LIN {X 0,Y 143.834,Z 840.119,A -85,B 0,C 180,E1 -24449.132,E2 -24449.132} C_VEL
LIN {X 0,Y 144.282,Z 844.837,A -85,B 0,C 180,E1 -24453.998,E2 -24453.998} C_VEL
LIN {X 0,Y 145.051,Z 847.23,A -85,B 0,C 180,E1 -24457.193,E2 -24457.193} C_VEL
LIN {X 0,Y 147.333,Z 850.158,A -85,B 0,C 180,E1 -24462.562,E2 -24462.562} C_VEL
LIN {X 0,Y 150.85,Z 851.632,A -85,B 0,C 180,E1 -24468.065,E2 -24468.065} C_VEL
LIN {X 0,Y 155.654,Z 851.525,A -85,B 0,C 180,E1 -24473.384,E2 -24473.384} C_VEL
LIN {X 0,Y 161.705,Z 849.693,A -85,B 0,C 180,E1 -24478.445,E2 -24478.445} C_VEL
LIN {X 0,Y 168.926,Z 846.027,A -85,B 0,C 180,E1 -24483.134,E2 -24483.134} C_VEL
LIN {X 0,Y 175.939,Z 841.345,A -85,B 0,C 180,E1 -24486.882,E2 -24486.882} C_VEL
LIN {X 0,Y 182.747,Z 835.741,A -85,B 0,C 180,E1 -24489.966,E2 -24489.966} C_VEL
LIN {X 0,Y 184.593,Z 833.905,A -85,B 0,C 180,E1 -24490.974,E2 -24490.974} C_VEL
LIN {X 0,Y 185.748,Z 831.879,A -85,B 0,C 180,E1 -24493.121,E2 -24493.121} C_VEL
LIN {X 0,Y 186.699,Z 829.958,A -85,B 0,C 180,E1 -24495.278,E2 -24495.278} C_VEL
LIN {X 0,Y 186.772,Z 828.948,A -85,B 0,C 180,E1 -24497.519,E2 -24497.519} C_VEL
LIN {X 0,Y 186.523,Z 828.401,A -85,B 0,C 180,E1 -24499.823,E2 -24499.823} C_VEL
LIN {X 0,Y 186.294,Z 828.27,A -85,B 0,C 180,E1 -24502.164,E2 -24502.164} C_VEL
LIN {X 0,Y 185.911,Z 829.094,A -85,B 0,C 180,E1 -24506.977,E2 -24506.977} C_VEL
LIN {X 0,Y 185.613,Z 830.4,A -85,B 0,C 180,E1 -24509.487,E2 -24509.487} C_VEL
LIN {X 0,Y 185.359,Z 832.163,A -85,B 0,C 180,E1 -24512.061,E2 -24512.061} C_VEL
LIN {X 0,Y 184.447,Z 837.377,A -85,B 0,C 180,E1 -24516.853,E2 -24516.853} C_VEL
LIN {X 0,Y 183.603,Z 840.183,A -85,B 0,C 180,E1 -24518.656,E2 -24518.656} C_VEL
LIN {X 0,Y 178.489,Z 848.812,A -85,B 0,C 180,E1 -24522.398,E2 -24522.398} C_VEL
LIN {X 0,Y 172.641,Z 857.248,A -85,B 0,C 180,E1 -24526.207,E2 -24526.207} C_VEL
LIN {X 0,Y 167.309,Z 863.837,A -85,B 0,C 180,E1 -24529.478,E2 -24529.478} C_VEL
LIN {X 0,Y 160.39,Z 870.953,A -85,B 0,C 180,E1 -24533.733,E2 -24533.733} C_VEL
LIN {X 0,Y 155.765,Z 875.456,A -85,B 0,C 180,E1 -24537.218,E2 -24537.218} C_VEL
LIN {X 0,Y 150.033,Z 880.097,A -85,B 0,C 180,E1 -24542.067,E2 -24542.067} C_VEL
LIN {X 0,Y 145.757,Z 883.409,A -85,B 0,C 180,E1 -24547.31,E2 -24547.31} C_VEL
LIN {X 0,Y 143.255,Z 885.452,A -85,B 0,C 180,E1 -24552.881,E2 -24552.881} C_VEL
LIN {X 0,Y 142.332,Z 886.187,A -85,B 0,C 180,E1 -24558.608,E2 -24558.608} C_VEL
LIN {X 0,Y 142.891,Z 885.548,A -85,B 0,C 180,E1 -24564.354,E2 -24564.354} C_VEL
LIN {X 0,Y 143.6,Z 884.69,A -85,B 0,C 180,E1 -24567.194,E2 -24567.194} C_VEL
LIN {X 0,Y 144.38,Z 883.383,A -85,B 0,C 180,E1 -24570,E2 -24570} C_VEL
LIN {X 0,Y 143.787,Z 880.036,A -85,B 0,C 180,E1 -24574.204,E2 -24574.204} C_VEL
LIN {X 0,Y 143.334,Z 875.413,A -85,B 0,C 180,E1 -24578.458,E2 -24578.458} C_VEL
LIN {X 0,Y 143.531,Z 869.496,A -85,B 0,C 180,E1 -24582.727,E2 -24582.727} C_VEL
LIN {X 0,Y 144.492,Z 862.057,A -85,B 0,C 180,E1 -24586.968,E2 -24586.968} C_VEL
LIN {X 0,Y 145.758,Z 854.433,A -85,B 0,C 180,E1 -24590.461,E2 -24590.461} C_VEL
LIN {X 0,Y 146.006,Z 847.076,A -85,B 0,C 180,E1 -24593.254,E2 -24593.254} C_VEL
LIN {X 0,Y 146.09,Z 837.104,A -85,B 0,C 180,E1 -24596.423,E2 -24596.423} C_VEL
LIN {X 0,Y 146.295,Z 825.525,A -85,B 0,C 180,E1 -24599.451,E2 -24599.451} C_VEL
LIN {X 0,Y 146.225,Z 812.879,A -85,B 0,C 180,E1 -24602.12,E2 -24602.12} C_VEL
LIN {X 0,Y 146.168,Z 798.933,A -85,B 0,C 180,E1 -24604.399,E2 -24604.399} C_VEL
LIN {X 0,Y 145.863,Z 785.037,A -85,B 0,C 180,E1 -24606.066,E2 -24606.066} C_VEL
LIN {X 0,Y 145.877,Z 782.396,A -85,B 0,C 180,E1 -24606.383,E2 -24606.383} C_VEL
LIN {X 0,Y 147.213,Z 778.09,A -85,B 0,C 180,E1 -24610.196,E2 -24610.196} C_VEL
LIN {X 0,Y 146.718,Z 774.986,A -85,B 0,C 180,E1 -24612.994,E2 -24612.994} C_VEL
LIN {X 0,Y 146.278,Z 773.253,A -85,B 0,C 180,E1 -24614.614,E2 -24614.614} C_VEL
LIN {X 0,Y 145.108,Z 771.082,A -85,B 0,C 180,E1 -24616.721,E2 -24616.721} C_VEL
LIN {X 0,Y 141.527,Z 767.841,A -85,B 0,C 180,E1 -24620.183,E2 -24620.183} C_VEL
LIN {X 0,Y 137.462,Z 764.026,A -85,B 0,C 180,E1 -24624.571,E2 -24624.571} C_VEL
LIN {X 0,Y 136.858,Z 762.629,A -85,B 0,C 180,E1 -24626.117,E2 -24626.117} C_VEL
LIN {X 0,Y 136.237,Z 759.516,A -85,B 0,C 180,E1 -24629.629,E2 -24629.629} C_VEL
LIN {X 0,Y 136.082,Z 759.532,A -85,B 0,C 180,E1 -24635.596,E2 -24635.596} C_VEL
LIN {X 0,Y 136.243,Z 759.512,A -85,B 0,C 180,E1 -24638.833,E2 -24638.833} C_VEL
LIN {X 0,Y 136.269,Z 759.51,A -85,B 0,C 180,E1 -24645.056,E2 -24645.056} C_VEL
LIN {X 0,Y 136.446,Z 759.487,A -85,B 0,C 180,E1 -24648.138,E2 -24648.138} C_VEL
LIN {X 0,Y 136.552,Z 759.471,A -85,B 0,C 180,E1 -24651.118,E2 -24651.118} C_VEL
LIN {X 0,Y 137.131,Z 759.397,A -85,B 0,C 180,E1 -24660,E2 -24660} C_VEL
LIN {X 0,Y 136.548,Z 759.471,A -85,B 0,C 180,E1 -24668.883,E2 -24668.883} C_VEL
LIN {X 0,Y 136.418,Z 759.491,A -85,B 0,C 180,E1 -24671.893,E2 -24671.893} C_VEL
LIN {X 0,Y 136.19,Z 759.517,A -85,B 0,C 180,E1 -24678.037,E2 -24678.037} C_VEL
LIN {X 0,Y 136.159,Z 759.523,A -85,B 0,C 180,E1 -24681.707,E2 -24681.707} C_VEL
LIN {X 0,Y 136.062,Z 759.535,A -85,B 0,C 180,E1 -24688.586,E2 -24688.586} C_VEL
LIN {X 0,Y 136.04,Z 759.534,A -85,B 0,C 180,E1 -24694.631,E2 -24694.631} C_VEL
LIN {X 0,Y 136.025,Z 759.541,A -85,B 0,C 180,E1 -24699.195,E2 -24699.195} C_VEL
LIN {X 0,Y 135.978,Z 759.542,A -85,B 0,C 180,E1 -24703.649,E2 -24703.649} C_VEL
LIN {X 0,Y 135.983,Z 759.547,A -85,B 0,C 180,E1 -24707.788,E2 -24707.788} C_VEL
LIN {X 0,Y 136.021,Z 759.535,A -85,B 0,C 180,E1 -24711.682,E2 -24711.682} C_VEL
LIN {X 0,Y 136.051,Z 759.538,A -85,B 0,C 180,E1 -24715.743,E2 -24715.743} C_VEL
LIN {X 0,Y 136.084,Z 759.532,A -85,B 0,C 180,E1 -24722.303,E2 -24722.303} C_VEL
LIN {X 0,Y 136.183,Z 759.516,A -85,B 0,C 180,E1 -24728.823,E2 -24728.823} C_VEL
LIN {X 0,Y 136.232,Z 759.512,A -85,B 0,C 180,E1 -24735.052,E2 -24735.052} C_VEL
LIN {X 0,Y 136.427,Z 759.486,A -85,B 0,C 180,E1 -24738.178,E2 -24738.178} C_VEL
LIN {X 0,Y 136.538,Z 759.478,A -85,B 0,C 180,E1 -24741.117,E2 -24741.117} C_VEL
LIN {X 0,Y 137.114,Z 759.404,A -85,B 0,C 180,E1 -24750,E2 -24750} C_VEL
LIN {X 0,Y 136.54,Z 759.477,A -85,B 0,C 180,E1 -24758.883,E2 -24758.883} C_VEL
LIN {X 0,Y 136.443,Z 759.484,A -85,B 0,C 180,E1 -24761.89,E2 -24761.89} C_VEL
LIN {X 0,Y 136.241,Z 759.514,A -85,B 0,C 180,E1 -24768.03,E2 -24768.03} C_VEL
LIN {X 0,Y 136.198,Z 759.518,A -85,B 0,C 180,E1 -24771.746,E2 -24771.746} C_VEL
LIN {X 0,Y 136.143,Z 759.589,A -85,B 0,C 180,E1 -24777.372,E2 -24777.372} C_VEL
LIN {X 0,Y 140.03,Z 771.67,A -85,B 0,C 180,E1 -24780.126,E2 -24780.126} C_VEL
LIN {X 0,Y 142.873,Z 781.876,A -85,B 0,C 180,E1 -24782.759,E2 -24782.759} C_VEL
LIN {X 0,Y 145.205,Z 791.325,A -85,B 0,C 180,E1 -24785.508,E2 -24785.508} C_VEL
LIN {X 0,Y 143.314,Z 801.057,A -85,B 0,C 180,E1 -24788.313,E2 -24788.313} C_VEL
LIN {X 0,Y 141.097,Z 811.829,A -85,B 0,C 180,E1 -24792.148,E2 -24792.148} C_VEL
LIN {X 0,Y 139.253,Z 820.681,A -85,B 0,C 180,E1 -24796.055,E2 -24796.055} C_VEL
LIN {X 0,Y 137.705,Z 829.579,A -85,B 0,C 180,E1 -24800.977,E2 -24800.977} C_VEL
LIN {X 0,Y 136.942,Z 836.317,A -85,B 0,C 180,E1 -24805.63,E2 -24805.63} C_VEL
LIN {X 0,Y 136.771,Z 842.282,A -85,B 0,C 180,E1 -24810.875,E2 -24810.875} C_VEL
LIN {X 0,Y 137.795,Z 847.229,A -85,B 0,C 180,E1 -24816.646,E2 -24816.646} C_VEL
LIN {X 0,Y 138.634,Z 848.953,A -85,B 0,C 180,E1 -24819.215,E2 -24819.215} C_VEL
LIN {X 0,Y 140.099,Z 850.688,A -85,B 0,C 180,E1 -24822.483,E2 -24822.483} C_VEL
LIN {X 0,Y 143.626,Z 852.615,A -85,B 0,C 180,E1 -24828.142,E2 -24828.142} C_VEL
LIN {X 0,Y 148.497,Z 852.967,A -85,B 0,C 180,E1 -24833.663,E2 -24833.663} C_VEL
LIN {X 0,Y 154.647,Z 851.703,A -85,B 0,C 180,E1 -24838.885,E2 -24838.885} C_VEL
LIN {X 0,Y 161.987,Z 848.675,A -85,B 0,C 180,E1 -24843.723,E2 -24843.723} C_VEL
LIN {X 0,Y 168.479,Z 845.008,A -85,B 0,C 180,E1 -24847.189,E2 -24847.189} C_VEL
LIN {X 0,Y 175.411,Z 840.184,A -85,B 0,C 180,E1 -24850.387,E2 -24850.387} C_VEL
LIN {X 0,Y 177.834,Z 838.261,A -85,B 0,C 180,E1 -24851.396,E2 -24851.396} C_VEL
LIN {X 0,Y 179.375,Z 836.805,A -85,B 0,C 180,E1 -24852.444,E2 -24852.444} C_VEL
LIN {X 0,Y 181.164,Z 834.2,A -85,B 0,C 180,E1 -24855.757,E2 -24855.757} C_VEL
LIN {X 0,Y 181.291,Z 833.426,A -85,B 0,C 180,E1 -24858.067,E2 -24858.067} C_VEL
LIN {X 0,Y 181.084,Z 833.09,A -85,B 0,C 180,E1 -24861.336,E2 -24861.336} C_VEL
LIN {X 0,Y 180.8,Z 833.559,A -85,B 0,C 180,E1 -24865.315,E2 -24865.315} C_VEL
LIN {X 0,Y 180.552,Z 834.454,A -85,B 0,C 180,E1 -24867.846,E2 -24867.846} C_VEL
LIN {X 0,Y 180.088,Z 836.926,A -85,B 0,C 180,E1 -24871.791,E2 -24871.791} C_VEL
LIN {X 0,Y 179.045,Z 841.299,A -85,B 0,C 180,E1 -24876.071,E2 -24876.071} C_VEL
LIN {X 0,Y 178.556,Z 842.717,A -85,B 0,C 180,E1 -24877.121,E2 -24877.121} C_VEL
LIN {X 0,Y 177.052,Z 845.185,A -85,B 0,C 180,E1 -24878.374,E2 -24878.374} C_VEL
LIN {X 0,Y 172.35,Z 851.866,A -85,B 0,C 180,E1 -24881.527,E2 -24881.527} C_VEL
LIN {X 0,Y 166.626,Z 859.074,A -85,B 0,C 180,E1 -24885.049,E2 -24885.049} C_VEL
LIN {X 0,Y 160.162,Z 865.94,A -85,B 0,C 180,E1 -24888.836,E2 -24888.836} C_VEL
LIN {X 0,Y 152.993,Z 872.424,A -85,B 0,C 180,E1 -24893.331,E2 -24893.331} C_VEL
LIN {X 0,Y 148.206,Z 876.389,A -85,B 0,C 180,E1 -24896.952,E2 -24896.952} C_VEL
LIN {X 0,Y 143.769,Z 879.528,A -85,B 0,C 180,E1 -24900.735,E2 -24900.735} C_VEL
LIN {X 0,Y 139.194,Z 882.578,A -85,B 0,C 180,E1 -24906.176,E2 -24906.176} C_VEL
LIN {X 0,Y 136.457,Z 884.351,A -85,B 0,C 180,E1 -24911.999,E2 -24911.999} C_VEL
LIN {X 0,Y 135.388,Z 884.858,A -85,B 0,C 180,E1 -24918.016,E2 -24918.016} C_VEL
LIN {X 0,Y 135.913,Z 884.037,A -85,B 0,C 180,E1 -24924.064,E2 -24924.064} C_VEL
LIN {X 0,Y 136.642,Z 883.095,A -85,B 0,C 180,E1 -24927.051,E2 -24927.051} C_VEL
LIN {X 0,Y 137.433,Z 881.708,A -85,B 0,C 180,E1 -24930,E2 -24930} C_VEL
LIN {X 0,Y 136.786,Z 878.178,A -85,B 0,C 180,E1 -24934.42,E2 -24934.42} C_VEL
LIN {X 0,Y 136.358,Z 873.319,A -85,B 0,C 180,E1 -24938.895,E2 -24938.895} C_VEL
LIN {X 0,Y 136.677,Z 867.118,A -85,B 0,C 180,E1 -24943.379,E2 -24943.379} C_VEL
LIN {X 0,Y 137.766,Z 859.376,A -85,B 0,C 180,E1 -24947.823,E2 -24947.823} C_VEL
LIN {X 0,Y 138.728,Z 853.091,A -85,B 0,C 180,E1 -24950.77,E2 -24950.77} C_VEL
LIN {X 0,Y 138.939,Z 845.219,A -85,B 0,C 180,E1 -24953.87,E2 -24953.87} C_VEL
LIN {X 0,Y 139.02,Z 835.571,A -85,B 0,C 180,E1 -24957.064,E2 -24957.064} C_VEL
LIN {X 0,Y 139.267,Z 825.325,A -85,B 0,C 180,E1 -24959.89,E2 -24959.89} C_VEL
LIN {X 0,Y 139.253,Z 813.767,A -85,B 0,C 180,E1 -24962.53,E2 -24962.53} C_VEL
LIN {X 0,Y 139.325,Z 801.501,A -85,B 0,C 180,E1 -24964.752,E2 -24964.752} C_VEL
LIN {X 0,Y 139.138,Z 786.767,A -85,B 0,C 180,E1 -24966.77,E2 -24966.77} C_VEL
LIN {X 0,Y 139.045,Z 781.432,A -85,B 0,C 180,E1 -24967.339,E2 -24967.339} C_VEL
LIN {X 0,Y 140.139,Z 777.838,A -85,B 0,C 180,E1 -24970.689,E2 -24970.689} C_VEL
LIN {X 0,Y 139.098,Z 773.388,A -85,B 0,C 180,E1 -24975.02,E2 -24975.02} C_VEL
LIN {X 0,Y 137.813,Z 767.424,A -85,B 0,C 180,E1 -24981.015,E2 -24981.015} C_VEL
LIN {X 0,Y 136.858,Z 762.629,A -85,B 0,C 180,E1 -24986.117,E2 -24986.117} C_VEL
LIN {X 0,Y 136.276,Z 761.453,A -85,B 0,C 180,E1 -24987.665,E2 -24987.665} C_VEL
LIN {X 0,Y 135.267,Z 760.692,A -85,B 0,C 180,E1 -24989.234,E2 -24989.234} C_VEL
LIN {X 0,Y 132.644,Z 760.099,A -85,B 0,C 180,E1 -24992.426,E2 -24992.426} C_VEL
LIN {X 0,Y 129.364,Z 760.371,A -85,B 0,C 180,E1 -24997.546,E2 -24997.546} C_VEL
LIN {X 0,Y 129.079,Z 760.397,A -85,B 0,C 180,E1 -24999.332,E2 -24999.332} C_VEL
LIN {X 0,Y 129.194,Z 760.39,A -85,B 0,C 180,E1 -25004.217,E2 -25004.217} C_VEL
LIN {X 0,Y 129.367,Z 760.37,A -85,B 0,C 180,E1 -25007.923,E2 -25007.923} C_VEL
LIN {X 0,Y 129.478,Z 760.351,A -85,B 0,C 180,E1 -25010.629,E2 -25010.629} C_VEL
LIN {X 0,Y 130.086,Z 760.275,A -85,B 0,C 180,E1 -25020,E2 -25020} C_VEL
LIN {X 0,Y 129.471,Z 760.355,A -85,B 0,C 180,E1 -25029.373,E2 -25029.373} C_VEL
LIN {X 0,Y 129.301,Z 760.379,A -85,B 0,C 180,E1 -25032.558,E2 -25032.558} C_VEL
LIN {X 0,Y 129.104,Z 760.402,A -85,B 0,C 180,E1 -25039.064,E2 -25039.064} C_VEL
LIN {X 0,Y 129.073,Z 760.405,A -85,B 0,C 180,E1 -25042.405,E2 -25042.405} C_VEL
LIN {X 0,Y 129,Z 760.417,A -85,B 0,C 180,E1 -25049.363,E2 -25049.363} C_VEL
LIN {X 0,Y 128.956,Z 760.417,A -85,B 0,C 180,E1 -25055.166,E2 -25055.166} C_VEL
LIN {X 0,Y 128.923,Z 760.422,A -85,B 0,C 180,E1 -25060.857,E2 -25060.857} C_VEL
LIN {X 0,Y 128.912,Z 760.425,A -85,B 0,C 180,E1 -25065.132,E2 -25065.132} C_VEL
LIN {X 0,Y 128.934,Z 760.42,A -85,B 0,C 180,E1 -25069.741,E2 -25069.741} C_VEL
LIN {X 0,Y 128.955,Z 760.421,A -85,B 0,C 180,E1 -25074.835,E2 -25074.835} C_VEL
LIN {X 0,Y 128.982,Z 760.414,A -85,B 0,C 180,E1 -25080.671,E2 -25080.671} C_VEL
LIN {X 0,Y 129.068,Z 760.402,A -85,B 0,C 180,E1 -25087.773,E2 -25087.773} C_VEL
LIN {X 0,Y 129.153,Z 760.396,A -85,B 0,C 180,E1 -25094.212,E2 -25094.212} C_VEL
LIN {X 0,Y 129.346,Z 760.367,A -85,B 0,C 180,E1 -25097.97,E2 -25097.97} C_VEL
LIN {X 0,Y 129.464,Z 760.358,A -85,B 0,C 180,E1 -25100.628,E2 -25100.628} C_VEL
LIN {X 0,Y 130.069,Z 760.282,A -85,B 0,C 180,E1 -25110,E2 -25110} C_VEL
LIN {X 0,Y 129.466,Z 760.359,A -85,B 0,C 180,E1 -25119.373,E2 -25119.373} C_VEL
LIN {X 0,Y 129.346,Z 760.366,A -85,B 0,C 180,E1 -25122.553,E2 -25122.553} C_VEL
LIN {X 0,Y 129.153,Z 760.396,A -85,B 0,C 180,E1 -25129.057,E2 -25129.057} C_VEL
LIN {X 0,Y 129.11,Z 760.402,A -85,B 0,C 180,E1 -25132.399,E2 -25132.399} C_VEL
LIN {X 0,Y 129.082,Z 760.407,A -85,B 0,C 180,E1 -25136.256,E2 -25136.256} C_VEL
LIN {X 0,Y 133.457,Z 774.164,A -85,B 0,C 180,E1 -25139.703,E2 -25139.703} C_VEL
LIN {X 0,Y 136.415,Z 785.069,A -85,B 0,C 180,E1 -25142.749,E2 -25142.749} C_VEL
LIN {X 0,Y 138.166,Z 792.115,A -85,B 0,C 180,E1 -25144.926,E2 -25144.926} C_VEL
LIN {X 0,Y 136.285,Z 801.745,A -85,B 0,C 180,E1 -25147.831,E2 -25147.831} C_VEL
LIN {X 0,Y 134.074,Z 812.127,A -85,B 0,C 180,E1 -25151.671,E2 -25151.671} C_VEL
LIN {X 0,Y 132.011,Z 821.956,A -85,B 0,C 180,E1 -25156.203,E2 -25156.203} C_VEL
LIN {X 0,Y 130.623,Z 829.9,A -85,B 0,C 180,E1 -25160.787,E2 -25160.787} C_VEL
LIN {X 0,Y 129.827,Z 836.713,A -85,B 0,C 180,E1 -25165.678,E2 -25165.678} C_VEL
LIN {X 0,Y 129.673,Z 842.464,A -85,B 0,C 180,E1 -25170.805,E2 -25170.805} C_VEL
LIN {X 0,Y 130.554,Z 847.211,A -85,B 0,C 180,E1 -25176.228,E2 -25176.228} C_VEL
LIN {X 0,Y 132.8,Z 851.058,A -85,B 0,C 180,E1 -25182.289,E2 -25182.289} C_VEL
LIN {X 0,Y 136.391,Z 853.453,A -85,B 0,C 180,E1 -25188.251,E2 -25188.251} C_VEL
LIN {X 0,Y 141.333,Z 854.283,A -85,B 0,C 180,E1 -25194.01,E2 -25194.01} C_VEL
LIN {X 0,Y 144.856,Z 854.056,A -85,B 0,C 180,E1 -25197.219,E2 -25197.219} C_VEL
LIN {X 0,Y 148.402,Z 853.339,A -85,B 0,C 180,E1 -25200,E2 -25200} C_VEL
LIN {X 0,Y 155.062,Z 851.131,A -85,B 0,C 180,E1 -25204.338,E2 -25204.338} C_VEL
LIN {X 0,Y 160.892,Z 848.401,A -85,B 0,C 180,E1 -25207.53,E2 -25207.53} C_VEL
LIN {X 0,Y 168.027,Z 844.247,A -85,B 0,C 180,E1 -25210.849,E2 -25210.849} C_VEL
LIN {X 0,Y 173.086,Z 840.715,A -85,B 0,C 180,E1 -25212.964,E2 -25212.964} C_VEL
LIN {X 0,Y 174.171,Z 839.71,A -85,B 0,C 180,E1 -25214.011,E2 -25214.011} C_VEL
LIN {X 0,Y 175.47,Z 838.269,A -85,B 0,C 180,E1 -25216.282,E2 -25216.282} C_VEL
LIN {X 0,Y 175.639,Z 837.702,A -85,B 0,C 180,E1 -25218.669,E2 -25218.669} C_VEL
LIN {X 0,Y 175.61,Z 837.57,A -85,B 0,C 180,E1 -25221.111,E2 -25221.111} C_VEL
LIN {X 0,Y 175.441,Z 837.835,A -85,B 0,C 180,E1 -25223.615,E2 -25223.615} C_VEL
LIN {X 0,Y 175.378,Z 838.414,A -85,B 0,C 180,E1 -25226.155,E2 -25226.155} C_VEL
LIN {X 0,Y 174.956,Z 839.705,A -85,B 0,C 180,E1 -25228.819,E2 -25228.819} C_VEL
LIN {X 0,Y 174.346,Z 842.006,A -85,B 0,C 180,E1 -25232.164,E2 -25232.164} C_VEL
LIN {X 0,Y 173.232,Z 845.59,A -85,B 0,C 180,E1 -25235.766,E2 -25235.766} C_VEL
LIN {X 0,Y 172.669,Z 846.605,A -85,B 0,C 180,E1 -25236.498,E2 -25236.498} C_VEL
LIN {X 0,Y 167.576,Z 853.056,A -85,B 0,C 180,E1 -25239.741,E2 -25239.741} C_VEL
LIN {X 0,Y 160.676,Z 860.68,A -85,B 0,C 180,E1 -25243.803,E2 -25243.803} C_VEL
LIN {X 0,Y 154.848,Z 866.146,A -85,B 0,C 180,E1 -25247.094,E2 -25247.094} C_VEL
LIN {X 0,Y 147.294,Z 872.302,A -85,B 0,C 180,E1 -25251.663,E2 -25251.663} C_VEL
LIN {X 0,Y 142.274,Z 875.971,A -85,B 0,C 180,E1 -25255.383,E2 -25255.383} C_VEL
LIN {X 0,Y 137.606,Z 878.897,A -85,B 0,C 180,E1 -25259.287,E2 -25259.287} C_VEL
LIN {X 0,Y 132.695,Z 881.659,A -85,B 0,C 180,E1 -25264.931,E2 -25264.931} C_VEL
LIN {X 0,Y 129.701,Z 883.21,A -85,B 0,C 180,E1 -25271.027,E2 -25271.027} C_VEL
LIN {X 0,Y 128.474,Z 883.509,A -85,B 0,C 180,E1 -25277.36,E2 -25277.36} C_VEL
LIN {X 0,Y 128.929,Z 882.497,A -85,B 0,C 180,E1 -25283.741,E2 -25283.741} C_VEL
LIN {X 0,Y 129.7,Z 881.428,A -85,B 0,C 180,E1 -25286.893,E2 -25286.893} C_VEL
LIN {X 0,Y 130.496,Z 879.906,A -85,B 0,C 180,E1 -25290,E2 -25290} C_VEL
LIN {X 0,Y 129.816,Z 876.146,A -85,B 0,C 180,E1 -25294.658,E2 -25294.658} C_VEL
LIN {X 0,Y 129.407,Z 871.063,A -85,B 0,C 180,E1 -25299.377,E2 -25299.377} C_VEL
LIN {X 0,Y 129.8,Z 864.633,A -85,B 0,C 180,E1 -25304.102,E2 -25304.102} C_VEL
LIN {X 0,Y 131.05,Z 856.614,A -85,B 0,C 180,E1 -25308.77,E2 -25308.77} C_VEL
LIN {X 0,Y 131.685,Z 851.726,A -85,B 0,C 180,E1 -25311.115,E2 -25311.115} C_VEL
LIN {X 0,Y 131.961,Z 841.558,A -85,B 0,C 180,E1 -25315.218,E2 -25315.218} C_VEL
LIN {X 0,Y 132.094,Z 831.268,A -85,B 0,C 180,E1 -25318.61,E2 -25318.61} C_VEL
LIN {X 0,Y 132.226,Z 819.666,A -85,B 0,C 180,E1 -25321.743,E2 -25321.743} C_VEL
LIN {X 0,Y 132.4,Z 806.647,A -85,B 0,C 180,E1 -25324.562,E2 -25324.562} C_VEL
LIN {X 0,Y 132.409,Z 792.821,A -85,B 0,C 180,E1 -25326.841,E2 -25326.841} C_VEL
LIN {X 0,Y 132.283,Z 780.454,A -85,B 0,C 180,E1 -25328.405,E2 -25328.405} C_VEL
LIN {X 0,Y 133.013,Z 778.141,A -85,B 0,C 180,E1 -25330.683,E2 -25330.683} C_VEL
LIN {X 0,Y 131.752,Z 772.841,A -85,B 0,C 180,E1 -25336.096,E2 -25336.096} C_VEL
LIN {X 0,Y 130.611,Z 767.537,A -85,B 0,C 180,E1 -25341.772,E2 -25341.772} C_VEL
LIN {X 0,Y 129.661,Z 762.733,A -85,B 0,C 180,E1 -25347.178,E2 -25347.178} C_VEL
LIN {X 0,Y 129.168,Z 760.394,A -85,B 0,C 180,E1 -25350.076,E2 -25350.076} C_VEL
LIN {X 0,Y 129.107,Z 760.403,A -85,B 0,C 180,E1 -25357.729,E2 -25357.729} C_VEL
LIN {X 0,Y 129.079,Z 760.397,A -85,B 0,C 180,E1 -25359.332,E2 -25359.332} C_VEL
LIN {X 0,Y 128.48,Z 760.476,A -85,B 0,C 180,E1 -25361.941,E2 -25361.941} C_VEL
LIN {X 0,Y 127.007,Z 760.666,A -85,B 0,C 180,E1 -25364.523,E2 -25364.523} C_VEL
LIN {X 0,Y 122.724,Z 761.206,A -85,B 0,C 180,E1 -25371.647,E2 -25371.647} C_VEL
LIN {X 0,Y 122.423,Z 761.233,A -85,B 0,C 180,E1 -25373.525,E2 -25373.525} C_VEL
LIN {X 0,Y 123.04,Z 761.152,A -85,B 0,C 180,E1 -25380,E2 -25380} C_VEL
LIN {X 0,Y 122.406,Z 761.231,A -85,B 0,C 180,E1 -25386.802,E2 -25386.802} C_VEL
LIN {X 0,Y 122.29,Z 761.252,A -85,B 0,C 180,E1 -25392.315,E2 -25392.315} C_VEL
LIN {X 0,Y 122.076,Z 761.271,A -85,B 0,C 180,E1 -25396.73,E2 -25396.73} C_VEL
LIN {X 0,Y 122.003,Z 761.287,A -85,B 0,C 180,E1 -25402.827,E2 -25402.827} C_VEL
LIN {X 0,Y 121.915,Z 761.298,A -85,B 0,C 180,E1 -25410.152,E2 -25410.152} C_VEL
LIN {X 0,Y 121.88,Z 761.302,A -85,B 0,C 180,E1 -25416.169,E2 -25416.169} C_VEL
LIN {X 0,Y 121.863,Z 761.3,A -85,B 0,C 180,E1 -25421.434,E2 -25421.434} C_VEL
LIN {X 0,Y 121.863,Z 761.303,A -85,B 0,C 180,E1 -25428.567,E2 -25428.567} C_VEL
LIN {X 0,Y 121.907,Z 761.299,A -85,B 0,C 180,E1 -25434.795,E2 -25434.795} C_VEL
LIN {X 0,Y 121.904,Z 761.293,A -85,B 0,C 180,E1 -25439.859,E2 -25439.859} C_VEL
LIN {X 0,Y 121.98,Z 761.285,A -85,B 0,C 180,E1 -25447.2,E2 -25447.2} C_VEL
LIN {X 0,Y 122.065,Z 761.279,A -85,B 0,C 180,E1 -25453.269,E2 -25453.269} C_VEL
LIN {X 0,Y 122.289,Z 761.246,A -85,B 0,C 180,E1 -25457.691,E2 -25457.691} C_VEL
LIN {X 0,Y 122.392,Z 761.238,A -85,B 0,C 180,E1 -25460.081,E2 -25460.081} C_VEL
LIN {X 0,Y 122.561,Z 761.212,A -85,B 0,C 180,E1 -25466.713,E2 -25466.713} C_VEL
LIN {X 0,Y 123.023,Z 761.16,A -85,B 0,C 180,E1 -25470,E2 -25470} C_VEL
LIN {X 0,Y 122.408,Z 761.234,A -85,B 0,C 180,E1 -25476.594,E2 -25476.594} C_VEL
LIN {X 0,Y 122.404,Z 761.236,A -85,B 0,C 180,E1 -25479.919,E2 -25479.919} C_VEL
LIN {X 0,Y 122.241,Z 761.251,A -85,B 0,C 180,E1 -25483.296,E2 -25483.296} C_VEL
LIN {X 0,Y 122.045,Z 761.278,A -85,B 0,C 180,E1 -25490.214,E2 -25490.214} C_VEL
LIN {X 0,Y 122.019,Z 761.337,A -85,B 0,C 180,E1 -25495.251,E2 -25495.251} C_VEL
LIN {X 0,Y 125.928,Z 773.313,A -85,B 0,C 180,E1 -25498.32,E2 -25498.32} C_VEL
LIN {X 0,Y 128.763,Z 783.441,A -85,B 0,C 180,E1 -25501.233,E2 -25501.233} C_VEL
LIN {X 0,Y 131.116,Z 792.785,A -85,B 0,C 180,E1 -25504.251,E2 -25504.251} C_VEL
LIN {X 0,Y 130.535,Z 796.757,A -85,B 0,C 180,E1 -25505.456,E2 -25505.456} C_VEL
LIN {X 0,Y 128.121,Z 807.666,A -85,B 0,C 180,E1 -25509.21,E2 -25509.21} C_VEL
LIN {X 0,Y 125.922,Z 817.566,A -85,B 0,C 180,E1 -25513.484,E2 -25513.484} C_VEL
LIN {X 0,Y 124.147,Z 826.513,A -85,B 0,C 180,E1 -25518.304,E2 -25518.304} C_VEL
LIN {X 0,Y 122.952,Z 835.002,A -85,B 0,C 180,E1 -25524.09,E2 -25524.09} C_VEL
LIN {X 0,Y 122.56,Z 841.158,A -85,B 0,C 180,E1 -25529.334,E2 -25529.334} C_VEL
LIN {X 0,Y 123.053,Z 845.921,A -85,B 0,C 180,E1 -25534.392,E2 -25534.392} C_VEL
LIN {X 0,Y 124.702,Z 850.184,A -85,B 0,C 180,E1 -25540.235,E2 -25540.235} C_VEL
LIN {X 0,Y 126.345,Z 852.21,A -85,B 0,C 180,E1 -25543.851,E2 -25543.851} C_VEL
LIN {X 0,Y 129.133,Z 854.139,A -85,B 0,C 180,E1 -25548.421,E2 -25548.421} C_VEL
LIN {X 0,Y 134.175,Z 855.467,A -85,B 0,C 180,E1 -25554.394,E2 -25554.394} C_VEL
LIN {X 0,Y 137.002,Z 855.561,A -85,B 0,C 180,E1 -25557.059,E2 -25557.059} C_VEL
LIN {X 0,Y 140.561,Z 855.217,A -85,B 0,C 180,E1 -25560,E2 -25560} C_VEL
LIN {X 0,Y 148.169,Z 853.406,A -85,B 0,C 180,E1 -25565.067,E2 -25565.067} C_VEL
LIN {X 0,Y 156.838,Z 849.881,A -85,B 0,C 180,E1 -25569.652,E2 -25569.652} C_VEL
LIN {X 0,Y 164.784,Z 845.539,A -85,B 0,C 180,E1 -25573.108,E2 -25573.108} C_VEL
LIN {X 0,Y 168.113,Z 843.414,A -85,B 0,C 180,E1 -25574.527,E2 -25574.527} C_VEL
LIN {X 0,Y 169.611,Z 842.139,A -85,B 0,C 180,E1 -25576.861,E2 -25576.861} C_VEL
LIN {X 0,Y 169.85,Z 841.812,A -85,B 0,C 180,E1 -25579.331,E2 -25579.331} C_VEL
LIN {X 0,Y 169.845,Z 841.87,A -85,B 0,C 180,E1 -25581.864,E2 -25581.864} C_VEL
LIN {X 0,Y 169.74,Z 842.34,A -85,B 0,C 180,E1 -25584.459,E2 -25584.459} C_VEL
LIN {X 0,Y 169.544,Z 843.227,A -85,B 0,C 180,E1 -25587.128,E2 -25587.128} C_VEL
LIN {X 0,Y 168.793,Z 845.739,A -85,B 0,C 180,E1 -25591.363,E2 -25591.363} C_VEL
LIN {X 0,Y 167.406,Z 849.131,A -85,B 0,C 180,E1 -25595.05,E2 -25595.05} C_VEL
LIN {X 0,Y 162.919,Z 854.114,A -85,B 0,C 180,E1 -25597.839,E2 -25597.839} C_VEL
LIN {X 0,Y 157.778,Z 859.334,A -85,B 0,C 180,E1 -25600.778,E2 -25600.778} C_VEL
LIN {X 0,Y 151.486,Z 864.916,A -85,B 0,C 180,E1 -25604.266,E2 -25604.266} C_VEL
LIN {X 0,Y 143.647,Z 870.799,A -85,B 0,C 180,E1 -25608.662,E2 -25608.662} C_VEL
LIN {X 0,Y 136.463,Z 875.557,A -85,B 0,C 180,E1 -25613.682,E2 -25613.682} C_VEL
LIN {X 0,Y 131.533,Z 878.243,A -85,B 0,C 180,E1 -25617.702,E2 -25617.702} C_VEL
LIN {X 0,Y 126.268,Z 880.746,A -85,B 0,C 180,E1 -25623.559,E2 -25623.559} C_VEL
LIN {X 0,Y 122.991,Z 882.025,A -85,B 0,C 180,E1 -25629.949,E2 -25629.949} C_VEL
LIN {X 0,Y 121.588,Z 882.079,A -85,B 0,C 180,E1 -25636.631,E2 -25636.631} C_VEL
LIN {X 0,Y 121.981,Z 880.842,A -85,B 0,C 180,E1 -25643.383,E2 -25643.383} C_VEL
LIN {X 0,Y 122.744,Z 879.708,A -85,B 0,C 180,E1 -25646.717,E2 -25646.717} C_VEL
LIN {X 0,Y 123.567,Z 878.115,A -85,B 0,C 180,E1 -25650,E2 -25650} C_VEL
LIN {X 0,Y 122.8,Z 874.104,A -85,B 0,C 180,E1 -25654.924,E2 -25654.924} C_VEL
LIN {X 0,Y 122.479,Z 868.779,A -85,B 0,C 180,E1 -25659.912,E2 -25659.912} C_VEL
LIN {X 0,Y 122.951,Z 862.001,A -85,B 0,C 180,E1 -25664.905,E2 -25664.905} C_VEL
LIN {X 0,Y 124.369,Z 853.603,A -85,B 0,C 180,E1 -25669.819,E2 -25669.819} C_VEL
LIN {X 0,Y 124.731,Z 847.336,A -85,B 0,C 180,E1 -25672.791,E2 -25672.791} C_VEL
LIN {X 0,Y 124.846,Z 837.357,A -85,B 0,C 180,E1 -25676.766,E2 -25676.766} C_VEL
LIN {X 0,Y 125.13,Z 826.403,A -85,B 0,C 180,E1 -25680.364,E2 -25680.364} C_VEL
LIN {X 0,Y 125.292,Z 813.869,A -85,B 0,C 180,E1 -25683.677,E2 -25683.677} C_VEL
LIN {X 0,Y 125.561,Z 800.328,A -85,B 0,C 180,E1 -25686.492,E2 -25686.492} C_VEL
LIN {X 0,Y 125.539,Z 785.881,A -85,B 0,C 180,E1 -25688.725,E2 -25688.725} C_VEL
LIN {X 0,Y 125.532,Z 779.441,A -85,B 0,C 180,E1 -25689.554,E2 -25689.554} C_VEL
LIN {X 0,Y 125.828,Z 778.051,A -85,B 0,C 180,E1 -25691.016,E2 -25691.016} C_VEL
LIN {X 0,Y 124.367,Z 772.256,A -85,B 0,C 180,E1 -25697.303,E2 -25697.303} C_VEL
LIN {X 0,Y 123.332,Z 767.338,A -85,B 0,C 180,E1 -25702.919,E2 -25702.919} C_VEL
LIN {X 0,Y 122.371,Z 762.373,A -85,B 0,C 180,E1 -25708.877,E2 -25708.877} C_VEL
LIN {X 0,Y 122.091,Z 761.274,A -85,B 0,C 180,E1 -25710.522,E2 -25710.522} C_VEL
LIN {X 0,Y 122.023,Z 761.284,A -85,B 0,C 180,E1 -25717.15,E2 -25717.15} C_VEL
LIN {X 0,Y 122.109,Z 761.271,A -85,B 0,C 180,E1 -25723.275,E2 -25723.275} C_VEL
LIN {X 0,Y 122.318,Z 761.247,A -85,B 0,C 180,E1 -25727.624,E2 -25727.624} C_VEL
LIN {X 0,Y 122.424,Z 761.234,A -85,B 0,C 180,E1 -25733.407,E2 -25733.407} C_VEL
LIN {X 0,Y 122.423,Z 761.233,A -85,B 0,C 180,E1 -25733.525,E2 -25733.525} C_VEL
LIN {X 0,Y 121.751,Z 761.319,A -85,B 0,C 180,E1 -25736.277,E2 -25736.277} C_VEL
LIN {X 0,Y 120.183,Z 761.511,A -85,B 0,C 180,E1 -25738.995,E2 -25738.995} C_VEL
LIN {X 0,Y 115.63,Z 762.077,A -85,B 0,C 180,E1 -25746.525,E2 -25746.525} C_VEL
LIN {X 0,Y 115.285,Z 762.113,A -85,B 0,C 180,E1 -25748.523,E2 -25748.523} C_VEL
LIN {X 0,Y 115.207,Z 762.134,A -85,B 0,C 180,E1 -25752.566,E2 -25752.566} C_VEL
LIN {X 0,Y 114.979,Z 762.159,A -85,B 0,C 180,E1 -25757.796,E2 -25757.796} C_VEL
LIN {X 0,Y 114.916,Z 762.166,A -85,B 0,C 180,E1 -25763.457,E2 -25763.457} C_VEL
LIN {X 0,Y 114.847,Z 762.179,A -85,B 0,C 180,E1 -25771.05,E2 -25771.05} C_VEL
LIN {X 0,Y 114.775,Z 762.189,A -85,B 0,C 180,E1 -25777.759,E2 -25777.759} C_VEL
LIN {X 0,Y 114.778,Z 762.181,A -85,B 0,C 180,E1 -25782.712,E2 -25782.712} C_VEL
LIN {X 0,Y 114.786,Z 762.187,A -85,B 0,C 180,E1 -25787.663,E2 -25787.663} C_VEL
LIN {X 0,Y 114.783,Z 762.185,A -85,B 0,C 180,E1 -25792.748,E2 -25792.748} C_VEL
LIN {X 0,Y 114.839,Z 762.173,A -85,B 0,C 180,E1 -25798.958,E2 -25798.958} C_VEL
LIN {X 0,Y 114.894,Z 762.169,A -85,B 0,C 180,E1 -25806.571,E2 -25806.571} C_VEL
LIN {X 0,Y 114.968,Z 762.164,A -85,B 0,C 180,E1 -25812.203,E2 -25812.203} C_VEL
LIN {X 0,Y 115.307,Z 762.121,A -85,B 0,C 180,E1 -25819.464,E2 -25819.464} C_VEL
LIN {X 0,Y 115.487,Z 762.092,A -85,B 0,C 180,E1 -25826.511,E2 -25826.511} C_VEL
LIN {X 0,Y 115.975,Z 762.038,A -85,B 0,C 180,E1 -25830,E2 -25830} C_VEL
LIN {X 0,Y 115.352,Z 762.114,A -85,B 0,C 180,E1 -25836.999,E2 -25836.999} C_VEL
LIN {X 0,Y 115.25,Z 762.122,A -85,B 0,C 180,E1 -25842.657,E2 -25842.657} C_VEL
LIN {X 0,Y 115.011,Z 762.159,A -85,B 0,C 180,E1 -25847.791,E2 -25847.791} C_VEL
LIN {X 0,Y 114.962,Z 762.165,A -85,B 0,C 180,E1 -25854.016,E2 -25854.016} C_VEL
LIN {X 0,Y 119.219,Z 775.253,A -85,B 0,C 180,E1 -25857.661,E2 -25857.661} C_VEL
LIN {X 0,Y 122.28,Z 786.47,A -85,B 0,C 180,E1 -25861.15,E2 -25861.15} C_VEL
LIN {X 0,Y 124.16,Z 794.75,A -85,B 0,C 180,E1 -25863.985,E2 -25863.985} C_VEL
LIN {X 0,Y 121.581,Z 806.071,A -85,B 0,C 180,E1 -25867.878,E2 -25867.878} C_VEL
LIN {X 0,Y 119.126,Z 816.675,A -85,B 0,C 180,E1 -25872.484,E2 -25872.484} C_VEL
LIN {X 0,Y 117.123,Z 826.48,A -85,B 0,C 180,E1 -25877.885,E2 -25877.885} C_VEL
LIN {X 0,Y 115.893,Z 834.896,A -85,B 0,C 180,E1 -25883.753,E2 -25883.753} C_VEL
LIN {X 0,Y 115.488,Z 841.588,A -85,B 0,C 180,E1 -25889.663,E2 -25889.663} C_VEL
LIN {X 0,Y 116.091,Z 846.659,A -85,B 0,C 180,E1 -25895.243,E2 -25895.243} C_VEL
LIN {X 0,Y 117.645,Z 850.549,A -85,B 0,C 180,E1 -25900.598,E2 -25900.598} C_VEL
LIN {X 0,Y 120.547,Z 853.817,A -85,B 0,C 180,E1 -25906.514,E2 -25906.514} C_VEL
LIN {X 0,Y 122.953,Z 855.255,A -85,B 0,C 180,E1 -25910.126,E2 -25910.126} C_VEL
LIN {X 0,Y 127.018,Z 856.489,A -85,B 0,C 180,E1 -25914.852,E2 -25914.852} C_VEL
LIN {X 0,Y 133.543,Z 856.741,A -85,B 0,C 180,E1 -25920.682,E2 -25920.682} C_VEL
LIN {X 0,Y 141.306,Z 855.494,A -85,B 0,C 180,E1 -25925.886,E2 -25925.886} C_VEL
LIN {X 0,Y 150.13,Z 852.59,A -85,B 0,C 180,E1 -25930.555,E2 -25930.555} C_VEL
LIN {X 0,Y 158.279,Z 848.876,A -85,B 0,C 180,E1 -25934.097,E2 -25934.097} C_VEL
LIN {X 0,Y 161.098,Z 847.337,A -85,B 0,C 180,E1 -25935.174,E2 -25935.174} C_VEL
LIN {X 0,Y 163.629,Z 845.785,A -85,B 0,C 180,E1 -25937.497,E2 -25937.497} C_VEL
LIN {X 0,Y 163.883,Z 845.731,A -85,B 0,C 180,E1 -25940.064,E2 -25940.064} C_VEL
LIN {X 0,Y 163.869,Z 845.975,A -85,B 0,C 180,E1 -25942.705,E2 -25942.705} C_VEL
LIN {X 0,Y 163.73,Z 846.768,A -85,B 0,C 180,E1 -25945.655,E2 -25945.655} C_VEL
LIN {X 0,Y 163.39,Z 847.882,A -85,B 0,C 180,E1 -25948.239,E2 -25948.239} C_VEL
LIN {X 0,Y 162.731,Z 849.718,A -85,B 0,C 180,E1 -25951.215,E2 -25951.215} C_VEL
LIN {X 0,Y 161.347,Z 852.34,A -85,B 0,C 180,E1 -25954.145,E2 -25954.145} C_VEL
LIN {X 0,Y 155.232,Z 858.063,A -85,B 0,C 180,E1 -25957.599,E2 -25957.599} C_VEL
LIN {X 0,Y 148.93,Z 863.338,A -85,B 0,C 180,E1 -25960.97,E2 -25960.97} C_VEL
LIN {X 0,Y 142.53,Z 867.936,A -85,B 0,C 180,E1 -25964.358,E2 -25964.358} C_VEL
LIN {X 0,Y 134.429,Z 872.999,A -85,B 0,C 180,E1 -25969.193,E2 -25969.193} C_VEL
LIN {X 0,Y 128.971,Z 875.961,A -85,B 0,C 180,E1 -25973.171,E2 -25973.171} C_VEL
LIN {X 0,Y 122.556,Z 878.779,A -85,B 0,C 180,E1 -25978.928,E2 -25978.928} C_VEL
LIN {X 0,Y 117.923,Z 880.403,A -85,B 0,C 180,E1 -25985.342,E2 -25985.342} C_VEL
LIN {X 0,Y 115.305,Z 880.84,A -85,B 0,C 180,E1 -25992.256,E2 -25992.256} C_VEL
LIN {X 0,Y 114.66,Z 880.078,A -85,B 0,C 180,E1 -25999.404,E2 -25999.404} C_VEL
LIN {X 0,Y 115.813,Z 877.916,A -85,B 0,C 180,E1 -26006.521,E2 -26006.521} C_VEL
LIN {X 0,Y 116.626,Z 876.173,A -85,B 0,C 180,E1 -26010,E2 -26010} C_VEL
LIN {X 0,Y 115.832,Z 871.944,A -85,B 0,C 180,E1 -26015.221,E2 -26015.221} C_VEL
LIN {X 0,Y 115.556,Z 866.366,A -85,B 0,C 180,E1 -26020.513,E2 -26020.513} C_VEL
LIN {X 0,Y 116.171,Z 859.324,A -85,B 0,C 180,E1 -26025.797,E2 -26025.797} C_VEL
LIN {X 0,Y 117.411,Z 852.135,A -85,B 0,C 180,E1 -26030.132,E2 -26030.132} C_VEL
LIN {X 0,Y 117.704,Z 843.695,A -85,B 0,C 180,E1 -26034.236,E2 -26034.236} C_VEL
LIN {X 0,Y 117.871,Z 833.034,A -85,B 0,C 180,E1 -26038.489,E2 -26038.489} C_VEL
LIN {X 0,Y 118.114,Z 822.754,A -85,B 0,C 180,E1 -26041.876,E2 -26041.876} C_VEL
LIN {X 0,Y 118.478,Z 810.317,A -85,B 0,C 180,E1 -26045.218,E2 -26045.218} C_VEL
LIN {X 0,Y 118.707,Z 796.538,A -85,B 0,C 180,E1 -26048.071,E2 -26048.071} C_VEL
LIN {X 0,Y 118.789,Z 782.598,A -85,B 0,C 180,E1 -26050.217,E2 -26050.217} C_VEL
LIN {X 0,Y 118.682,Z 778.441,A -85,B 0,C 180,E1 -26050.786,E2 -26050.786} C_VEL
LIN {X 0,Y 117.621,Z 774.048,A -85,B 0,C 180,E1 -26055.808,E2 -26055.808} C_VEL
LIN {X 0,Y 116.29,Z 768.214,A -85,B 0,C 180,E1 -26062.818,E2 -26062.818} C_VEL
LIN {X 0,Y 115.273,Z 763.041,A -85,B 0,C 180,E1 -26069.408,E2 -26069.408} C_VEL
LIN {X 0,Y 115.026,Z 762.154,A -85,B 0,C 180,E1 -26070.739,E2 -26070.739} C_VEL
LIN {X 0,Y 114.979,Z 762.161,A -85,B 0,C 180,E1 -26078.485,E2 -26078.485} C_VEL
LIN {X 0,Y 115.134,Z 762.143,A -85,B 0,C 180,E1 -26085.868,E2 -26085.868} C_VEL
LIN {X 0,Y 115.325,Z 762.114,A -85,B 0,C 180,E1 -26089.466,E2 -26089.466} C_VEL
LIN {X 0,Y 115.52,Z 762.094,A -85,B 0,C 180,E1 -26096.512,E2 -26096.512} C_VEL
LIN {X 0,Y 115.991,Z 762.03,A -85,B 0,C 180,E1 -26100,E2 -26100} C_VEL
LIN {X 0,Y 115.285,Z 762.113,A -85,B 0,C 180,E1 -26108.523,E2 -26108.523} C_VEL
LIN {X 0,Y 114.574,Z 762.213,A -85,B 0,C 180,E1 -26111.436,E2 -26111.436} C_VEL
LIN {X 0,Y 112.976,Z 762.414,A -85,B 0,C 180,E1 -26114.315,E2 -26114.315} C_VEL
LIN {X 0,Y 108.243,Z 763.001,A -85,B 0,C 180,E1 -26122.306,E2 -26122.306} C_VEL
LIN {X 0,Y 107.798,Z 763.049,A -85,B 0,C 180,E1 -26124.437,E2 -26124.437} C_VEL
LIN {X 0,Y 107.773,Z 763.056,A -85,B 0,C 180,E1 -26132.033,E2 -26132.033} C_VEL
LIN {X 0,Y 107.683,Z 763.071,A -85,B 0,C 180,E1 -26138.447,E2 -26138.447} C_VEL
LIN {X 0,Y 107.67,Z 763.073,A -85,B 0,C 180,E1 -26145.891,E2 -26145.891} C_VEL
LIN {X 0,Y 107.682,Z 763.063,A -85,B 0,C 180,E1 -26151.555,E2 -26151.555} C_VEL
LIN {X 0,Y 107.777,Z 763.053,A -85,B 0,C 180,E1 -26158.556,E2 -26158.556} C_VEL
LIN {X 0,Y 107.863,Z 763.044,A -85,B 0,C 180,E1 -26166.987,E2 -26166.987} C_VEL
LIN {X 0,Y 107.864,Z 763.048,A -85,B 0,C 180,E1 -26170.987,E2 -26170.987} C_VEL
LIN {X 0,Y 108.207,Z 763.002,A -85,B 0,C 180,E1 -26178.764,E2 -26178.764} C_VEL
LIN {X 0,Y 108.289,Z 762.996,A -85,B 0,C 180,E1 -26182.542,E2 -26182.542} C_VEL
LIN {X 0,Y 108.9,Z 762.919,A -85,B 0,C 180,E1 -26190,E2 -26190} C_VEL
LIN {X 0,Y 108.293,Z 762.995,A -85,B 0,C 180,E1 -26197.458,E2 -26197.458} C_VEL
LIN {X 0,Y 108.171,Z 763.003,A -85,B 0,C 180,E1 -26202.948,E2 -26202.948} C_VEL
LIN {X 0,Y 107.927,Z 763.04,A -85,B 0,C 180,E1 -26211.99,E2 -26211.99} C_VEL
LIN {X 0,Y 107.949,Z 763.121,A -85,B 0,C 180,E1 -26212.741,E2 -26212.741} C_VEL
LIN {X 0,Y 111.698,Z 774.672,A -85,B 0,C 180,E1 -26216.132,E2 -26216.132} C_VEL
LIN {X 0,Y 114.849,Z 785.764,A -85,B 0,C 180,E1 -26219.764,E2 -26219.764} C_VEL
LIN {X 0,Y 117.188,Z 795.147,A -85,B 0,C 180,E1 -26223.178,E2 -26223.178} C_VEL
LIN {X 0,Y 114.308,Z 807.581,A -85,B 0,C 180,E1 -26227.698,E2 -26227.698} C_VEL
LIN {X 0,Y 112.055,Z 817.173,A -85,B 0,C 180,E1 -26232.103,E2 -26232.103} C_VEL
LIN {X 0,Y 110.295,Z 825.379,A -85,B 0,C 180,E1 -26236.764,E2 -26236.764} C_VEL
LIN {X 0,Y 108.959,Z 833.461,A -85,B 0,C 180,E1 -26242.445,E2 -26242.445} C_VEL
LIN {X 0,Y 108.385,Z 840.704,A -85,B 0,C 180,E1 -26248.751,E2 -26248.751} C_VEL
LIN {X 0,Y 109.133,Z 847.235,A -85,B 0,C 180,E1 -26255.995,E2 -26255.995} C_VEL
LIN {X 0,Y 110.929,Z 851.376,A -85,B 0,C 180,E1 -26261.869,E2 -26261.869} C_VEL
LIN {X 0,Y 114.614,Z 855.114,A -85,B 0,C 180,E1 -26268.846,E2 -26268.846} C_VEL
LIN {X 0,Y 119.861,Z 857.345,A -85,B 0,C 180,E1 -26275.417,E2 -26275.417} C_VEL
LIN {X 0,Y 126.546,Z 858.115,A -85,B 0,C 180,E1 -26281.445,E2 -26281.445} C_VEL
LIN {X 0,Y 134.487,Z 857.371,A -85,B 0,C 180,E1 -26286.828,E2 -26286.828} C_VEL
LIN {X 0,Y 143.483,Z 855.119,A -85,B 0,C 180,E1 -26291.582,E2 -26291.582} C_VEL
LIN {X 0,Y 150.926,Z 852.329,A -85,B 0,C 180,E1 -26294.841,E2 -26294.841} C_VEL
LIN {X 0,Y 153.723,Z 851.073,A -85,B 0,C 180,E1 -26295.921,E2 -26295.921} C_VEL
LIN {X 0,Y 157.524,Z 849.252,A -85,B 0,C 180,E1 -26298.198,E2 -26298.198} C_VEL
LIN {X 0,Y 157.736,Z 849.426,A -85,B 0,C 180,E1 -26300.882,E2 -26300.882} C_VEL
LIN {X 0,Y 157.712,Z 849.927,A -85,B 0,C 180,E1 -26303.644,E2 -26303.644} C_VEL
LIN {X 0,Y 157.444,Z 850.967,A -85,B 0,C 180,E1 -26306.777,E2 -26306.777} C_VEL
LIN {X 0,Y 156.982,Z 852.338,A -85,B 0,C 180,E1 -26309.502,E2 -26309.502} C_VEL
LIN {X 0,Y 156.353,Z 853.577,A -85,B 0,C 180,E1 -26311.345,E2 -26311.345} C_VEL
LIN {X 0,Y 155.586,Z 854.802,A -85,B 0,C 180,E1 -26312.823,E2 -26312.823} C_VEL
LIN {X 0,Y 148.706,Z 860.4,A -85,B 0,C 180,E1 -26316.539,E2 -26316.539} C_VEL
LIN {X 0,Y 141.591,Z 865.479,A -85,B 0,C 180,E1 -26320.186,E2 -26320.186} C_VEL
LIN {X 0,Y 133.23,Z 870.452,A -85,B 0,C 180,E1 -26324.59,E2 -26324.59} C_VEL
LIN {X 0,Y 127.119,Z 873.614,A -85,B 0,C 180,E1 -26328.436,E2 -26328.436} C_VEL
LIN {X 0,Y 119.738,Z 876.772,A -85,B 0,C 180,E1 -26334.059,E2 -26334.059} C_VEL
LIN {X 0,Y 113.694,Z 878.704,A -85,B 0,C 180,E1 -26340.361,E2 -26340.361} C_VEL
LIN {X 0,Y 109.785,Z 879.481,A -85,B 0,C 180,E1 -26347.412,E2 -26347.412} C_VEL
LIN {X 0,Y 107.922,Z 879.061,A -85,B 0,C 180,E1 -26354.901,E2 -26354.901} C_VEL
LIN {X 0,Y 108.119,Z 877.404,A -85,B 0,C 180,E1 -26362.53,E2 -26362.53} C_VEL
LIN {X 0,Y 108.917,Z 876.059,A -85,B 0,C 180,E1 -26366.3,E2 -26366.3} C_VEL
LIN {X 0,Y 109.716,Z 874.2,A -85,B 0,C 180,E1 -26370,E2 -26370} C_VEL
LIN {X 0,Y 108.848,Z 869.692,A -85,B 0,C 180,E1 -26375.557,E2 -26375.557} C_VEL
LIN {X 0,Y 108.664,Z 863.838,A -85,B 0,C 180,E1 -26381.188,E2 -26381.188} C_VEL
LIN {X 0,Y 109.471,Z 856.461,A -85,B 0,C 180,E1 -26386.792,E2 -26386.792} C_VEL
LIN {X 0,Y 110.423,Z 850.542,A -85,B 0,C 180,E1 -26390.49,E2 -26390.49} C_VEL
LIN {X 0,Y 110.647,Z 841.91,A -85,B 0,C 180,E1 -26394.885,E2 -26394.885} C_VEL
LIN {X 0,Y 110.902,Z 830.666,A -85,B 0,C 180,E1 -26399.556,E2 -26399.556} C_VEL
LIN {X 0,Y 111.234,Z 818.794,A -85,B 0,C 180,E1 -26403.562,E2 -26403.562} C_VEL
LIN {X 0,Y 111.643,Z 805.86,A -85,B 0,C 180,E1 -26407.009,E2 -26407.009} C_VEL
LIN {X 0,Y 111.969,Z 793.275,A -85,B 0,C 180,E1 -26409.638,E2 -26409.638} C_VEL
LIN {X 0,Y 111.901,Z 779.969,A -85,B 0,C 180,E1 -26411.731,E2 -26411.731} C_VEL
LIN {X 0,Y 111.326,Z 777.344,A -85,B 0,C 180,E1 -26412.29,E2 -26412.29} C_VEL
LIN {X 0,Y 109.669,Z 770.913,A -85,B 0,C 180,E1 -26420.264,E2 -26420.264} C_VEL
LIN {X 0,Y 108.717,Z 766.472,A -85,B 0,C 180,E1 -26426.137,E2 -26426.137} C_VEL
LIN {X 0,Y 107.955,Z 763.035,A -85,B 0,C 180,E1 -26431.041,E2 -26431.041} C_VEL
LIN {X 0,Y 107.911,Z 763.043,A -85,B 0,C 180,E1 -26436.998,E2 -26436.998} C_VEL
LIN {X 0,Y 108.031,Z 763.028,A -85,B 0,C 180,E1 -26444.917,E2 -26444.917} C_VEL
LIN {X 0,Y 108.254,Z 762.996,A -85,B 0,C 180,E1 -26448.769,E2 -26448.769} C_VEL
LIN {X 0,Y 108.444,Z 762.976,A -85,B 0,C 180,E1 -26456.285,E2 -26456.285} C_VEL
LIN {X 0,Y 108.917,Z 762.911,A -85,B 0,C 180,E1 -26460,E2 -26460} C_VEL
LIN {X 0,Y 108.235,Z 762.991,A -85,B 0,C 180,E1 -26468.432,E2 -26468.432} C_VEL
LIN {X 0,Y 108.141,Z 763.015,A -85,B 0,C 180,E1 -26472.88,E2 -26472.88} C_VEL
LIN {X 0,Y 107.875,Z 763.046,A -85,B 0,C 180,E1 -26479.011,E2 -26479.011} C_VEL
LIN {X 0,Y 107.798,Z 763.049,A -85,B 0,C 180,E1 -26484.437,E2 -26484.437} C_VEL
LIN {X 0,Y 106.973,Z 763.158,A -85,B 0,C 180,E1 -26487.553,E2 -26487.553} C_VEL
LIN {X 0,Y 105.353,Z 763.361,A -85,B 0,C 180,E1 -26490.638,E2 -26490.638} C_VEL
LIN {X 0,Y 100.889,Z 763.918,A -85,B 0,C 180,E1 -26499.238,E2 -26499.238} C_VEL
LIN {X 0,Y 100.564,Z 763.947,A -85,B 0,C 180,E1 -26501.523,E2 -26501.523} C_VEL
LIN {X 0,Y 100.641,Z 763.948,A -85,B 0,C 180,E1 -26505.707,E2 -26505.707} C_VEL
LIN {X 0,Y 100.621,Z 763.942,A -85,B 0,C 180,E1 -26511.052,E2 -26511.052} C_VEL
LIN {X 0,Y 100.681,Z 763.942,A -85,B 0,C 180,E1 -26516.894,E2 -26516.894} C_VEL
LIN {X 0,Y 100.707,Z 763.939,A -85,B 0,C 180,E1 -26525.247,E2 -26525.247} C_VEL
LIN {X 0,Y 100.776,Z 763.927,A -85,B 0,C 180,E1 -26529.593,E2 -26529.593} C_VEL
LIN {X 0,Y 101.117,Z 763.883,A -85,B 0,C 180,E1 -26537.965,E2 -26537.965} C_VEL
LIN {X 0,Y 101.223,Z 763.876,A -85,B 0,C 180,E1 -26542.018,E2 -26542.018} C_VEL
LIN {X 0,Y 101.828,Z 763.8,A -85,B 0,C 180,E1 -26550,E2 -26550} C_VEL
LIN {X 0,Y 101.234,Z 763.875,A -85,B 0,C 180,E1 -26557.982,E2 -26557.982} C_VEL
LIN {X 0,Y 101.101,Z 763.884,A -85,B 0,C 180,E1 -26563.291,E2 -26563.291} C_VEL
LIN {X 0,Y 100.9,Z 764.075,A -85,B 0,C 180,E1 -26571.316,E2 -26571.316} C_VEL
LIN {X 0,Y 104.727,Z 775.797,A -85,B 0,C 180,E1 -26575.048,E2 -26575.048} C_VEL
LIN {X 0,Y 107.602,Z 785.826,A -85,B 0,C 180,E1 -26578.53,E2 -26578.53} C_VEL
LIN {X 0,Y 110.03,Z 795.658,A -85,B 0,C 180,E1 -26582.287,E2 -26582.287} C_VEL
LIN {X 0,Y 109.513,Z 798.913,A -85,B 0,C 180,E1 -26583.458,E2 -26583.458} C_VEL
LIN {X 0,Y 106.851,Z 809.87,A -85,B 0,C 180,E1 -26587.88,E2 -26587.88} C_VEL
LIN {X 0,Y 104.186,Z 820.768,A -85,B 0,C 180,E1 -26593.517,E2 -26593.517} C_VEL
LIN {X 0,Y 102.542,Z 829.124,A -85,B 0,C 180,E1 -26598.932,E2 -26598.932} C_VEL
LIN {X 0,Y 101.51,Z 836.897,A -85,B 0,C 180,E1 -26605.169,E2 -26605.169} C_VEL
LIN {X 0,Y 101.489,Z 844.285,A -85,B 0,C 180,E1 -26612.632,E2 -26612.632} C_VEL
LIN {X 0,Y 103.075,Z 850.076,A -85,B 0,C 180,E1 -26620.067,E2 -26620.067} C_VEL
LIN {X 0,Y 105.874,Z 854.046,A -85,B 0,C 180,E1 -26626.565,E2 -26626.565} C_VEL
LIN {X 0,Y 109.832,Z 856.874,A -85,B 0,C 180,E1 -26632.647,E2 -26632.647} C_VEL
LIN {X 0,Y 113.082,Z 858.166,A -85,B 0,C 180,E1 -26636.436,E2 -26636.436} C_VEL
LIN {X 0,Y 119.578,Z 859.331,A -85,B 0,C 180,E1 -26642.349,E2 -26642.349} C_VEL
LIN {X 0,Y 127.721,Z 859.091,A -85,B 0,C 180,E1 -26647.91,E2 -26647.91} C_VEL
LIN {X 0,Y 136.903,Z 857.429,A -85,B 0,C 180,E1 -26652.739,E2 -26652.739} C_VEL
LIN {X 0,Y 146.992,Z 854.208,A -85,B 0,C 180,E1 -26657.01,E2 -26657.01} C_VEL
LIN {X 0,Y 151.154,Z 852.572,A -85,B 0,C 180,E1 -26658.994,E2 -26658.994} C_VEL
LIN {X 0,Y 151.419,Z 852.893,A -85,B 0,C 180,E1 -26661.829,E2 -26661.829} C_VEL
LIN {X 0,Y 151.343,Z 853.663,A -85,B 0,C 180,E1 -26664.704,E2 -26664.704} C_VEL
LIN {X 0,Y 150.94,Z 854.868,A -85,B 0,C 180,E1 -26667.788,E2 -26667.788} C_VEL
LIN {X 0,Y 149.94,Z 856.791,A -85,B 0,C 180,E1 -26671.037,E2 -26671.037} C_VEL
LIN {X 0,Y 149.016,Z 857.64,A -85,B 0,C 180,E1 -26671.904,E2 -26671.904} C_VEL
LIN {X 0,Y 142.171,Z 862.378,A -85,B 0,C 180,E1 -26675.347,E2 -26675.347} C_VEL
LIN {X 0,Y 135.23,Z 866.602,A -85,B 0,C 180,E1 -26678.779,E2 -26678.779} C_VEL
LIN {X 0,Y 126.085,Z 871.235,A -85,B 0,C 180,E1 -26683.562,E2 -26683.562} C_VEL
LIN {X 0,Y 117.851,Z 874.672,A -85,B 0,C 180,E1 -26689.005,E2 -26689.005} C_VEL
LIN {X 0,Y 110.622,Z 876.899,A -85,B 0,C 180,E1 -26695.125,E2 -26695.125} C_VEL
LIN {X 0,Y 105.161,Z 877.969,A -85,B 0,C 180,E1 -26702.107,E2 -26702.107} C_VEL
LIN {X 0,Y 101.932,Z 877.917,A -85,B 0,C 180,E1 -26709.834,E2 -26709.834} C_VEL
LIN {X 0,Y 100.924,Z 876.691,A -85,B 0,C 180,E1 -26717.941,E2 -26717.941} C_VEL
LIN {X 0,Y 102.024,Z 874.128,A -85,B 0,C 180,E1 -26726.05,E2 -26726.05} C_VEL
LIN {X 0,Y 102.788,Z 872.137,A -85,B 0,C 180,E1 -26730,E2 -26730} C_VEL
LIN {X 0,Y 101.869,Z 867.355,A -85,B 0,C 180,E1 -26735.94,E2 -26735.94} C_VEL
LIN {X 0,Y 101.814,Z 861.187,A -85,B 0,C 180,E1 -26741.951,E2 -26741.951} C_VEL
LIN {X 0,Y 102.812,Z 853.499,A -85,B 0,C 180,E1 -26747.915,E2 -26747.915} C_VEL
LIN {X 0,Y 103.428,Z 848.827,A -85,B 0,C 180,E1 -26750.9,E2 -26750.9} C_VEL
LIN {X 0,Y 103.569,Z 839.966,A -85,B 0,C 180,E1 -26755.632,E2 -26755.632} C_VEL
LIN {X 0,Y 103.893,Z 828.905,A -85,B 0,C 180,E1 -26760.487,E2 -26760.487} C_VEL
LIN {X 0,Y 104.25,Z 818.207,A -85,B 0,C 180,E1 -26764.334,E2 -26764.334} C_VEL
LIN {X 0,Y 104.756,Z 805.241,A -85,B 0,C 180,E1 -26768.052,E2 -26768.052} C_VEL
LIN {X 0,Y 105.184,Z 792.227,A -85,B 0,C 180,E1 -26770.967,E2 -26770.967} C_VEL
LIN {X 0,Y 105.178,Z 781.397,A -85,B 0,C 180,E1 -26772.861,E2 -26772.861} C_VEL
LIN {X 0,Y 103.811,Z 776.175,A -85,B 0,C 180,E1 -26774.003,E2 -26774.003} C_VEL
LIN {X 0,Y 102.326,Z 770.36,A -85,B 0,C 180,E1 -26781.82,E2 -26781.82} C_VEL
LIN {X 0,Y 101.311,Z 765.579,A -85,B 0,C 180,E1 -26788.649,E2 -26788.649} C_VEL
LIN {X 0,Y 100.889,Z 763.914,A -85,B 0,C 180,E1 -26791.386,E2 -26791.386} C_VEL
LIN {X 0,Y 100.798,Z 763.926,A -85,B 0,C 180,E1 -26795.27,E2 -26795.27} C_VEL
LIN {X 0,Y 100.816,Z 763.925,A -85,B 0,C 180,E1 -26799.601,E2 -26799.601} C_VEL
LIN {X 0,Y 101.102,Z 763.891,A -85,B 0,C 180,E1 -26806.702,E2 -26806.702} C_VEL
LIN {X 0,Y 101.242,Z 763.869,A -85,B 0,C 180,E1 -26812.02,E2 -26812.02} C_VEL
LIN {X 0,Y 101.844,Z 763.792,A -85,B 0,C 180,E1 -26820,E2 -26820} C_VEL
LIN {X 0,Y 101.233,Z 763.867,A -85,B 0,C 180,E1 -26827.982,E2 -26827.982} C_VEL
LIN {X 0,Y 101.055,Z 763.896,A -85,B 0,C 180,E1 -26833.184,E2 -26833.184} C_VEL
LIN {X 0,Y 100.789,Z 763.93,A -85,B 0,C 180,E1 -26840.405,E2 -26840.405} C_VEL
LIN {X 0,Y 100.734,Z 763.929,A -85,B 0,C 180,E1 -26844.909,E2 -26844.909} C_VEL
LIN {X 0,Y 100.684,Z 763.936,A -85,B 0,C 180,E1 -26853.11,E2 -26853.11} C_VEL
LIN {X 0,Y 100.635,Z 763.947,A -85,B 0,C 180,E1 -26859.807,E2 -26859.807} C_VEL
LIN {X 0,Y 100.564,Z 763.947,A -85,B 0,C 180,E1 -26861.523,E2 -26861.523} C_VEL
LIN {X 0,Y 99.879,Z 764.042,A -85,B 0,C 180,E1 -26864.87,E2 -26864.87} C_VEL
LIN {X 0,Y 98.328,Z 764.235,A -85,B 0,C 180,E1 -26868.187,E2 -26868.187} C_VEL
LIN {X 0,Y 93.834,Z 764.795,A -85,B 0,C 180,E1 -26877.458,E2 -26877.458} C_VEL
LIN {X 0,Y 93.48,Z 764.827,A -85,B 0,C 180,E1 -26879.928,E2 -26879.928} C_VEL
LIN {X 0,Y 93.592,Z 764.828,A -85,B 0,C 180,E1 -26884.305,E2 -26884.305} C_VEL
LIN {X 0,Y 93.637,Z 764.814,A -85,B 0,C 180,E1 -26887.959,E2 -26887.959} C_VEL
LIN {X 0,Y 93.96,Z 764.773,A -85,B 0,C 180,E1 -26896.503,E2 -26896.503} C_VEL
LIN {X 0,Y 94.153,Z 764.757,A -85,B 0,C 180,E1 -26901.415,E2 -26901.415} C_VEL
LIN {X 0,Y 94.757,Z 764.681,A -85,B 0,C 180,E1 -26910,E2 -26910} C_VEL
LIN {X 0,Y 94.169,Z 764.755,A -85,B 0,C 180,E1 -26918.585,E2 -26918.585} C_VEL
LIN {X 0,Y 94.017,Z 764.766,A -85,B 0,C 180,E1 -26923.64,E2 -26923.64} C_VEL
LIN {X 0,Y 93.795,Z 764.798,A -85,B 0,C 180,E1 -26929.563,E2 -26929.563} C_VEL
LIN {X 0,Y 97.817,Z 776.914,A -85,B 0,C 180,E1 -26933.838,E2 -26933.838} C_VEL
LIN {X 0,Y 100.634,Z 786.793,A -85,B 0,C 180,E1 -26937.56,E2 -26937.56} C_VEL
LIN {X 0,Y 102.903,Z 796.15,A -85,B 0,C 180,E1 -26941.385,E2 -26941.385} C_VEL
LIN {X 0,Y 103.019,Z 797.458,A -85,B 0,C 180,E1 -26941.919,E2 -26941.919} C_VEL
LIN {X 0,Y 99.993,Z 809.528,A -85,B 0,C 180,E1 -26946.917,E2 -26946.917} C_VEL
LIN {X 0,Y 97.414,Z 819.74,A -85,B 0,C 180,E1 -26952.323,E2 -26952.323} C_VEL
LIN {X 0,Y 95.499,Z 828.982,A -85,B 0,C 180,E1 -26958.521,E2 -26958.521} C_VEL
LIN {X 0,Y 94.446,Z 836.645,A -85,B 0,C 180,E1 -26964.94,E2 -26964.94} C_VEL
LIN {X 0,Y 94.24,Z 842.598,A -85,B 0,C 180,E1 -26971.006,E2 -26971.006} C_VEL
LIN {X 0,Y 95.406,Z 848.612,A -85,B 0,C 180,E1 -26978.387,E2 -26978.387} C_VEL
LIN {X 0,Y 97.959,Z 853.249,A -85,B 0,C 180,E1 -26985.457,E2 -26985.457} C_VEL
LIN {X 0,Y 101.777,Z 856.682,A -85,B 0,C 180,E1 -26992.061,E2 -26992.061} C_VEL
LIN {X 0,Y 105.585,Z 858.612,A -85,B 0,C 180,E1 -26996.81,E2 -26996.81} C_VEL
LIN {X 0,Y 112.647,Z 860.351,A -85,B 0,C 180,E1 -27003.392,E2 -27003.392} C_VEL
LIN {X 0,Y 121.018,Z 860.639,A -85,B 0,C 180,E1 -27009.152,E2 -27009.152} C_VEL
LIN {X 0,Y 130.419,Z 859.53,A -85,B 0,C 180,E1 -27014.071,E2 -27014.071} C_VEL
LIN {X 0,Y 140.672,Z 856.955,A -85,B 0,C 180,E1 -27018.331,E2 -27018.331} C_VEL
LIN {X 0,Y 144.439,Z 855.738,A -85,B 0,C 180,E1 -27019.913,E2 -27019.913} C_VEL
LIN {X 0,Y 144.918,Z 856.175,A -85,B 0,C 180,E1 -27022.862,E2 -27022.862} C_VEL
LIN {X 0,Y 144.673,Z 857.18,A -85,B 0,C 180,E1 -27025.926,E2 -27025.926} C_VEL
LIN {X 0,Y 143.854,Z 858.768,A -85,B 0,C 180,E1 -27029.245,E2 -27029.245} C_VEL
LIN {X 0,Y 142.509,Z 859.95,A -85,B 0,C 180,E1 -27030.731,E2 -27030.731} C_VEL
LIN {X 0,Y 135.675,Z 864.003,A -85,B 0,C 180,E1 -27034.023,E2 -27034.023} C_VEL
LIN {X 0,Y 128.416,Z 867.729,A -85,B 0,C 180,E1 -27037.479,E2 -27037.479} C_VEL
LIN {X 0,Y 121.261,Z 870.82,A -85,B 0,C 180,E1 -27041.109,E2 -27041.109} C_VEL
LIN {X 0,Y 112.566,Z 873.955,A -85,B 0,C 180,E1 -27046.623,E2 -27046.623} C_VEL
LIN {X 0,Y 104.883,Z 875.891,A -85,B 0,C 180,E1 -27052.909,E2 -27052.909} C_VEL
LIN {X 0,Y 98.944,Z 876.668,A -85,B 0,C 180,E1 -27060.184,E2 -27060.184} C_VEL
LIN {X 0,Y 95.357,Z 876.358,A -85,B 0,C 180,E1 -27068.376,E2 -27068.376} C_VEL
LIN {X 0,Y 94.107,Z 874.876,A -85,B 0,C 180,E1 -27077.053,E2 -27077.053} C_VEL
LIN {X 0,Y 95.175,Z 872.087,A -85,B 0,C 180,E1 -27085.765,E2 -27085.765} C_VEL
LIN {X 0,Y 95.886,Z 869.956,A -85,B 0,C 180,E1 -27090,E2 -27090} C_VEL
LIN {X 0,Y 94.921,Z 864.892,A -85,B 0,C 180,E1 -27096.376,E2 -27096.376} C_VEL
LIN {X 0,Y 94.959,Z 858.445,A -85,B 0,C 180,E1 -27102.828,E2 -27102.828} C_VEL
LIN {X 0,Y 96.134,Z 850.366,A -85,B 0,C 180,E1 -27109.204,E2 -27109.204} C_VEL
LIN {X 0,Y 96.433,Z 845.241,A -85,B 0,C 180,E1 -27112.496,E2 -27112.496} C_VEL
LIN {X 0,Y 96.511,Z 836.108,A -85,B 0,C 180,E1 -27117.462,E2 -27117.462} C_VEL
LIN {X 0,Y 96.871,Z 826.663,A -85,B 0,C 180,E1 -27121.734,E2 -27121.734} C_VEL
LIN {X 0,Y 97.383,Z 814.691,A -85,B 0,C 180,E1 -27126.156,E2 -27126.156} C_VEL
LIN {X 0,Y 98.025,Z 802.354,A -85,B 0,C 180,E1 -27129.791,E2 -27129.791} C_VEL
LIN {X 0,Y 98.467,Z 789.284,A -85,B 0,C 180,E1 -27132.768,E2 -27132.768} C_VEL
LIN {X 0,Y 98.471,Z 782.824,A -85,B 0,C 180,E1 -27133.979,E2 -27133.979} C_VEL
LIN {X 0,Y 96.278,Z 775.109,A -85,B 0,C 180,E1 -27135.789,E2 -27135.789} C_VEL
LIN {X 0,Y 94.981,Z 769.705,A -85,B 0,C 180,E1 -27143.705,E2 -27143.705} C_VEL
LIN {X 0,Y 93.922,Z 765.077,A -85,B 0,C 180,E1 -27150.897,E2 -27150.897} C_VEL
LIN {X 0,Y 93.825,Z 764.79,A -85,B 0,C 180,E1 -27152.085,E2 -27152.085} C_VEL
LIN {X 0,Y 93.698,Z 764.814,A -85,B 0,C 180,E1 -27157.974,E2 -27157.974} C_VEL
LIN {X 0,Y 94.067,Z 764.767,A -85,B 0,C 180,E1 -27167.048,E2 -27167.048} C_VEL
LIN {X 0,Y 94.175,Z 764.748,A -85,B 0,C 180,E1 -27171.417,E2 -27171.417} C_VEL
LIN {X 0,Y 94.773,Z 764.673,A -85,B 0,C 180,E1 -27180,E2 -27180} C_VEL
LIN {X 0,Y 94.163,Z 764.748,A -85,B 0,C 180,E1 -27188.585,E2 -27188.585} C_VEL
LIN {X 0,Y 93.964,Z 764.779,A -85,B 0,C 180,E1 -27193.511,E2 -27193.511} C_VEL
LIN {X 0,Y 93.66,Z 764.817,A -85,B 0,C 180,E1 -27202.037,E2 -27202.037} C_VEL
LIN {X 0,Y 93.595,Z 764.822,A -85,B 0,C 180,E1 -27206.779,E2 -27206.779} C_VEL
LIN {X 0,Y 93.582,Z 764.821,A -85,B 0,C 180,E1 -27214.3,E2 -27214.3} C_VEL
LIN {X 0,Y 93.528,Z 764.827,A -85,B 0,C 180,E1 -27222.555,E2 -27222.555} C_VEL
LIN {X 0,Y 93.531,Z 764.832,A -85,B 0,C 180,E1 -27228.714,E2 -27228.714} C_VEL
LIN {X 0,Y 93.58,Z 764.828,A -85,B 0,C 180,E1 -27235.703,E2 -27235.703} C_VEL
LIN {X 0,Y 93.48,Z 764.827,A -85,B 0,C 180,E1 -27239.928,E2 -27239.928} C_VEL
LIN {X 0,Y 92.759,Z 764.93,A -85,B 0,C 180,E1 -27243.526,E2 -27243.526} C_VEL
LIN {X 0,Y 91.205,Z 765.123,A -85,B 0,C 180,E1 -27247.098,E2 -27247.098} C_VEL
LIN {X 0,Y 87.091,Z 765.628,A -85,B 0,C 180,E1 -27257.137,E2 -27257.137} C_VEL
LIN {X 0,Y 86.975,Z 765.644,A -85,B 0,C 180,E1 -27259.795,E2 -27259.795} C_VEL
LIN {X 0,Y 87.687,Z 765.562,A -85,B 0,C 180,E1 -27270,E2 -27270} C_VEL
LIN {X 0,Y 87.079,Z 765.638,A -85,B 0,C 180,E1 -27279.29,E2 -27279.29} C_VEL
LIN {X 0,Y 86.933,Z 765.649,A -85,B 0,C 180,E1 -27284.037,E2 -27284.037} C_VEL
LIN {X 0,Y 86.775,Z 765.852,A -85,B 0,C 180,E1 -27287.834,E2 -27287.834} C_VEL
LIN {X 0,Y 90.67,Z 777.315,A -85,B 0,C 180,E1 -27292.202,E2 -27292.202} C_VEL
LIN {X 0,Y 93.513,Z 787.196,A -85,B 0,C 180,E1 -27296.203,E2 -27296.203} C_VEL
LIN {X 0,Y 96.023,Z 797.663,A -85,B 0,C 180,E1 -27300.82,E2 -27300.82} C_VEL
LIN {X 0,Y 93.395,Z 808.272,A -85,B 0,C 180,E1 -27305.378,E2 -27305.378} C_VEL
LIN {X 0,Y 90.7,Z 818.484,A -85,B 0,C 180,E1 -27310.93,E2 -27310.93} C_VEL
LIN {X 0,Y 88.518,Z 828.259,A -85,B 0,C 180,E1 -27317.69,E2 -27317.69} C_VEL
LIN {X 0,Y 87.389,Z 836.162,A -85,B 0,C 180,E1 -27324.564,E2 -27324.564} C_VEL
LIN {X 0,Y 87.26,Z 843.462,A -85,B 0,C 180,E1 -27332.371,E2 -27332.371} C_VEL
LIN {X 0,Y 88.407,Z 848.611,A -85,B 0,C 180,E1 -27339.041,E2 -27339.041} C_VEL
LIN {X 0,Y 91.15,Z 853.511,A -85,B 0,C 180,E1 -27346.625,E2 -27346.625} C_VEL
LIN {X 0,Y 95.266,Z 857.234,A -85,B 0,C 180,E1 -27353.646,E2 -27353.646} C_VEL
LIN {X 0,Y 100.651,Z 859.852,A -85,B 0,C 180,E1 -27360,E2 -27360} C_VEL
LIN {X 0,Y 105.76,Z 861.196,A -85,B 0,C 180,E1 -27364.588,E2 -27364.588} C_VEL
LIN {X 0,Y 114.496,Z 862.012,A -85,B 0,C 180,E1 -27370.611,E2 -27370.611} C_VEL
LIN {X 0,Y 124.015,Z 861.44,A -85,B 0,C 180,E1 -27375.547,E2 -27375.547} C_VEL
LIN {X 0,Y 134.471,Z 859.444,A -85,B 0,C 180,E1 -27379.819,E2 -27379.819} C_VEL
LIN {X 0,Y 137.481,Z 858.677,A -85,B 0,C 180,E1 -27380.967,E2 -27380.967} C_VEL
LIN {X 0,Y 138.186,Z 859.22,A -85,B 0,C 180,E1 -27384.008,E2 -27384.008} C_VEL
LIN {X 0,Y 137.676,Z 860.477,A -85,B 0,C 180,E1 -27387.35,E2 -27387.35} C_VEL
LIN {X 0,Y 136.726,Z 861.485,A -85,B 0,C 180,E1 -27389.091,E2 -27389.091} C_VEL
LIN {X 0,Y 129.209,Z 865.29,A -85,B 0,C 180,E1 -27392.532,E2 -27392.532} C_VEL
LIN {X 0,Y 121.631,Z 868.515,A -85,B 0,C 180,E1 -27396.007,E2 -27396.007} C_VEL
LIN {X 0,Y 111.938,Z 871.859,A -85,B 0,C 180,E1 -27401.112,E2 -27401.112} C_VEL
LIN {X 0,Y 103.261,Z 874.086,A -85,B 0,C 180,E1 -27407.108,E2 -27407.108} C_VEL
LIN {X 0,Y 95.822,Z 875.143,A -85,B 0,C 180,E1 -27414.072,E2 -27414.072} C_VEL
LIN {X 0,Y 90.565,Z 875.121,A -85,B 0,C 180,E1 -27422.25,E2 -27422.25} C_VEL
LIN {X 0,Y 87.766,Z 874.011,A -85,B 0,C 180,E1 -27431.318,E2 -27431.318} C_VEL
LIN {X 0,Y 87.561,Z 871.69,A -85,B 0,C 180,E1 -27440.762,E2 -27440.762} C_VEL
LIN {X 0,Y 88.802,Z 868.977,A -85,B 0,C 180,E1 -27447.732,E2 -27447.732} C_VEL
LIN {X 0,Y 88.957,Z 867.694,A -85,B 0,C 180,E1 -27450,E2 -27450} C_VEL
LIN {X 0,Y 87.989,Z 861.301,A -85,B 0,C 180,E1 -27458.035,E2 -27458.035} C_VEL
LIN {X 0,Y 88.364,Z 853.812,A -85,B 0,C 180,E1 -27465.344,E2 -27465.344} C_VEL
LIN {X 0,Y 89.201,Z 848.693,A -85,B 0,C 180,E1 -27469.442,E2 -27469.442} C_VEL
LIN {X 0,Y 89.402,Z 842.248,A -85,B 0,C 180,E1 -27473.758,E2 -27473.758} C_VEL
LIN {X 0,Y 89.624,Z 831.496,A -85,B 0,C 180,E1 -27479.723,E2 -27479.723} C_VEL
LIN {X 0,Y 90.068,Z 821.077,A -85,B 0,C 180,E1 -27484.452,E2 -27484.452} C_VEL
LIN {X 0,Y 90.766,Z 808.735,A -85,B 0,C 180,E1 -27488.942,E2 -27488.942} C_VEL
LIN {X 0,Y 91.47,Z 796.661,A -85,B 0,C 180,E1 -27492.418,E2 -27492.418} C_VEL
LIN {X 0,Y 91.933,Z 785.238,A -85,B 0,C 180,E1 -27494.998,E2 -27494.998} C_VEL
LIN {X 0,Y 88.769,Z 774.014,A -85,B 0,C 180,E1 -27497.896,E2 -27497.896} C_VEL
LIN {X 0,Y 87.588,Z 769.019,A -85,B 0,C 180,E1 -27505.829,E2 -27505.829} C_VEL
LIN {X 0,Y 86.802,Z 765.667,A -85,B 0,C 180,E1 -27511.589,E2 -27511.589} C_VEL
LIN {X 0,Y 86.647,Z 765.684,A -85,B 0,C 180,E1 -27521.069,E2 -27521.069} C_VEL
LIN {X 0,Y 86.931,Z 765.657,A -85,B 0,C 180,E1 -27525.964,E2 -27525.964} C_VEL
LIN {X 0,Y 87.085,Z 765.629,A -85,B 0,C 180,E1 -27530.712,E2 -27530.712} C_VEL
LIN {X 0,Y 87.702,Z 765.554,A -85,B 0,C 180,E1 -27540,E2 -27540} C_VEL
LIN {X 0,Y 87.066,Z 765.634,A -85,B 0,C 180,E1 -27549.291,E2 -27549.291} C_VEL
LIN {X 0,Y 86.861,Z 765.663,A -85,B 0,C 180,E1 -27554.048,E2 -27554.048} C_VEL
LIN {X 0,Y 86.607,Z 765.694,A -85,B 0,C 180,E1 -27558.941,E2 -27558.941} C_VEL
LIN {X 0,Y 86.563,Z 765.698,A -85,B 0,C 180,E1 -27566.737,E2 -27566.737} C_VEL
LIN {X 0,Y 86.501,Z 765.706,A -85,B 0,C 180,E1 -27575.662,E2 -27575.662} C_VEL
LIN {X 0,Y 86.451,Z 765.708,A -85,B 0,C 180,E1 -27582.976,E2 -27582.976} C_VEL
LIN {X 0,Y 86.453,Z 765.711,A -85,B 0,C 180,E1 -27589.433,E2 -27589.433} C_VEL
LIN {X 0,Y 86.524,Z 765.707,A -85,B 0,C 180,E1 -27595.349,E2 -27595.349} C_VEL
LIN {X 0,Y 86.523,Z 765.707,A -85,B 0,C 180,E1 -27603.317,E2 -27603.317} C_VEL
LIN {X 0,Y 86.592,Z 765.697,A -85,B 0,C 180,E1 -27611.056,E2 -27611.056} C_VEL
LIN {X 0,Y 86.864,Z 765.658,A -85,B 0,C 180,E1 -27616.147,E2 -27616.147} C_VEL
LIN {X 0,Y 86.975,Z 765.644,A -85,B 0,C 180,E1 -27619.795,E2 -27619.795} C_VEL
LIN {X 0,Y 86.826,Z 765.676,A -85,B 0,C 180,E1 -27622.38,E2 -27622.38} C_VEL
LIN {X 0,Y 85.63,Z 765.837,A -85,B 0,C 180,E1 -27626.232,E2 -27626.232} C_VEL
LIN {X 0,Y 82.466,Z 766.231,A -85,B 0,C 180,E1 -27632.763,E2 -27632.763} C_VEL
LIN {X 0,Y 80.335,Z 766.481,A -85,B 0,C 180,E1 -27638.363,E2 -27638.363} C_VEL
LIN {X 0,Y 79.886,Z 766.526,A -85,B 0,C 180,E1 -27641.285,E2 -27641.285} C_VEL
LIN {X 0,Y 79.793,Z 766.59,A -85,B 0,C 180,E1 -27645.649,E2 -27645.649} C_VEL
LIN {X 0,Y 83.901,Z 778.826,A -85,B 0,C 180,E1 -27650.856,E2 -27650.856} C_VEL
LIN {X 0,Y 86.972,Z 789.825,A -85,B 0,C 180,E1 -27655.744,E2 -27655.744} C_VEL
LIN {X 0,Y 88.97,Z 798.48,A -85,B 0,C 180,E1 -27659.884,E2 -27659.884} C_VEL
LIN {X 0,Y 86.762,Z 807.107,A -85,B 0,C 180,E1 -27663.799,E2 -27663.799} C_VEL
LIN {X 0,Y 83.765,Z 818.143,A -85,B 0,C 180,E1 -27670.039,E2 -27670.039} C_VEL
LIN {X 0,Y 81.631,Z 827.064,A -85,B 0,C 180,E1 -27676.467,E2 -27676.467} C_VEL
LIN {X 0,Y 80.369,Z 835.301,A -85,B 0,C 180,E1 -27683.823,E2 -27683.823} C_VEL
LIN {X 0,Y 80.196,Z 843.251,A -85,B 0,C 180,E1 -27692.703,E2 -27692.703} C_VEL
LIN {X 0,Y 81.727,Z 849.384,A -85,B 0,C 180,E1 -27701.074,E2 -27701.074} C_VEL
LIN {X 0,Y 85.691,Z 855.191,A -85,B 0,C 180,E1 -27710.559,E2 -27710.559} C_VEL
LIN {X 0,Y 91.389,Z 859.175,A -85,B 0,C 180,E1 -27718.683,E2 -27718.683} C_VEL
LIN {X 0,Y 98.927,Z 861.87,A -85,B 0,C 180,E1 -27725.953,E2 -27725.953} C_VEL
LIN {X 0,Y 107.83,Z 863.205,A -85,B 0,C 180,E1 -27732.133,E2 -27732.133} C_VEL
LIN {X 0,Y 117.943,Z 863.116,A -85,B 0,C 180,E1 -27737.334,E2 -27737.334} C_VEL
LIN {X 0,Y 130.339,Z 861.368,A -85,B 0,C 180,E1 -27742.175,E2 -27742.175} C_VEL
LIN {X 0,Y 131.321,Z 861.73,A -85,B 0,C 180,E1 -27744.52,E2 -27744.52} C_VEL
LIN {X 0,Y 130.307,Z 863.05,A -85,B 0,C 180,E1 -27747.607,E2 -27747.607} C_VEL
LIN {X 0,Y 121.919,Z 866.565,A -85,B 0,C 180,E1 -27751.252,E2 -27751.252} C_VEL
LIN {X 0,Y 112.368,Z 869.79,A -85,B 0,C 180,E1 -27755.601,E2 -27755.601} C_VEL
LIN {X 0,Y 102.663,Z 872.258,A -85,B 0,C 180,E1 -27761.146,E2 -27761.146} C_VEL
LIN {X 0,Y 93.998,Z 873.585,A -85,B 0,C 180,E1 -27767.707,E2 -27767.707} C_VEL
LIN {X 0,Y 86.979,Z 873.801,A -85,B 0,C 180,E1 -27775.554,E2 -27775.554} C_VEL
LIN {X 0,Y 82.474,Z 872.974,A -85,B 0,C 180,E1 -27784.781,E2 -27784.781} C_VEL
LIN {X 0,Y 80.664,Z 871.045,A -85,B 0,C 180,E1 -27794.847,E2 -27794.847} C_VEL
LIN {X 0,Y 81.556,Z 867.783,A -85,B 0,C 180,E1 -27805.056,E2 -27805.056} C_VEL
LIN {X 0,Y 82.071,Z 866.729,A -85,B 0,C 180,E1 -27807.546,E2 -27807.546} C_VEL
LIN {X 0,Y 82.02,Z 865.313,A -85,B 0,C 180,E1 -27809.999,E2 -27809.999} C_VEL
LIN {X 0,Y 81.123,Z 859.68,A -85,B 0,C 180,E1 -27817.466,E2 -27817.466} C_VEL
LIN {X 0,Y 81.418,Z 852.489,A -85,B 0,C 180,E1 -27825.008,E2 -27825.008} C_VEL
LIN {X 0,Y 82.26,Z 846.69,A -85,B 0,C 180,E1 -27829.983,E2 -27829.983} C_VEL
LIN {X 0,Y 82.342,Z 839.138,A -85,B 0,C 180,E1 -27835.261,E2 -27835.261} C_VEL
LIN {X 0,Y 82.683,Z 828.534,A -85,B 0,C 180,E1 -27841.413,E2 -27841.413} C_VEL
LIN {X 0,Y 83.287,Z 816.669,A -85,B 0,C 180,E1 -27846.958,E2 -27846.958} C_VEL
LIN {X 0,Y 84.1,Z 805.272,A -85,B 0,C 180,E1 -27851.228,E2 -27851.228} C_VEL
LIN {X 0,Y 84.947,Z 791.618,A -85,B 0,C 180,E1 -27855.176,E2 -27855.176} C_VEL
LIN {X 0,Y 85.095,Z 786.248,A -85,B 0,C 180,E1 -27856.47,E2 -27856.47} C_VEL
LIN {X 0,Y 81.284,Z 772.815,A -85,B 0,C 180,E1 -27860.42,E2 -27860.42} C_VEL
LIN {X 0,Y 80.239,Z 768.384,A -85,B 0,C 180,E1 -27868.297,E2 -27868.297} C_VEL
LIN {X 0,Y 79.756,Z 766.543,A -85,B 0,C 180,E1 -27871.785,E2 -27871.785} C_VEL
LIN {X 0,Y 79.529,Z 766.576,A -85,B 0,C 180,E1 -27879.3,E2 -27879.3} C_VEL
LIN {X 0,Y 79.825,Z 766.541,A -85,B 0,C 180,E1 -27885.573,E2 -27885.573} C_VEL
LIN {X 0,Y 79.968,Z 766.516,A -85,B 0,C 180,E1 -27889.877,E2 -27889.877} C_VEL
LIN {X 0,Y 80.632,Z 766.434,A -85,B 0,C 180,E1 -27900.001,E2 -27900.001} C_VEL
LIN {X 0,Y 79.943,Z 766.525,A -85,B 0,C 180,E1 -27910.127,E2 -27910.127} C_VEL
LIN {X 0,Y 79.69,Z 766.551,A -85,B 0,C 180,E1 -27915.342,E2 -27915.342} C_VEL
LIN {X 0,Y 79.482,Z 766.584,A -85,B 0,C 180,E1 -27920.714,E2 -27920.714} C_VEL
LIN {X 0,Y 79.464,Z 766.585,A -85,B 0,C 180,E1 -27927.82,E2 -27927.82} C_VEL
LIN {X 0,Y 79.368,Z 766.594,A -85,B 0,C 180,E1 -27932.094,E2 -27932.094} C_VEL
LIN {X 0,Y 79.362,Z 766.599,A -85,B 0,C 180,E1 -27938.309,E2 -27938.309} C_VEL
LIN {X 0,Y 79.382,Z 766.595,A -85,B 0,C 180,E1 -27945.096,E2 -27945.096} C_VEL
LIN {X 0,Y 79.382,Z 766.592,A -85,B 0,C 180,E1 -27952.828,E2 -27952.828} C_VEL
LIN {X 0,Y 79.34,Z 766.597,A -85,B 0,C 180,E1 -27957.895,E2 -27957.895} C_VEL
LIN {X 0,Y 79.47,Z 766.586,A -85,B 0,C 180,E1 -27963.757,E2 -27963.757} C_VEL
LIN {X 0,Y 79.462,Z 766.58,A -85,B 0,C 180,E1 -27969.282,E2 -27969.282} C_VEL
LIN {X 0,Y 79.788,Z 766.54,A -85,B 0,C 180,E1 -27975.681,E2 -27975.681} C_VEL
LIN {X 0,Y 79.934,Z 766.527,A -85,B 0,C 180,E1 -27979.873,E2 -27979.873} C_VEL
LIN {X 0,Y 80.616,Z 766.443,A -85,B 0,C 180,E1 -27990.001,E2 -27990.001} C_VEL
LIN {X 0,Y 79.886,Z 766.526,A -85,B 0,C 180,E1 -28001.285,E2 -28001.285} C_VEL
LIN {X 0,Y 79.777,Z 767.292,A -85,B 0,C 180,E1 -28003.338,E2 -28003.338} C_VEL
LIN {X 0,Y 79.661,Z 769.834,A -85,B 0,C 180,E1 -28005.614,E2 -28005.614} C_VEL
LIN {X 0,Y 79.526,Z 774.375,A -85,B 0,C 180,E1 -28007.817,E2 -28007.817} C_VEL
LIN {X 0,Y 79.483,Z 785.317,A -85,B 0,C 180,E1 -28011.964,E2 -28011.964} C_VEL
LIN {X 0,Y 80.273,Z 791.879,A -85,B 0,C 180,E1 -28014.981,E2 -28014.981} C_VEL
LIN {X 0,Y 81.976,Z 799.573,A -85,B 0,C 180,E1 -28019.015,E2 -28019.015} C_VEL
LIN {X 0,Y 78.879,Z 810.51,A -85,B 0,C 180,E1 -28024.495,E2 -28024.495} C_VEL
LIN {X 0,Y 75.742,Z 822.069,A -85,B 0,C 180,E1 -28032.07,E2 -28032.07} C_VEL
LIN {X 0,Y 73.651,Z 832.194,A -85,B 0,C 180,E1 -28040.908,E2 -28040.908} C_VEL
LIN {X 0,Y 72.992,Z 840.513,A -85,B 0,C 180,E1 -28050.063,E2 -28050.063} C_VEL
LIN {X 0,Y 74.128,Z 847.482,A -85,B 0,C 180,E1 -28059.408,E2 -28059.408} C_VEL
LIN {X 0,Y 77.652,Z 853.798,A -85,B 0,C 180,E1 -28069.571,E2 -28069.571} C_VEL
LIN {X 0,Y 82.477,Z 858.06,A -85,B 0,C 180,E1 -28077.56,E2 -28077.56} C_VEL
LIN {X 0,Y 88.715,Z 861.226,A -85,B 0,C 180,E1 -28084.543,E2 -28084.543} C_VEL
LIN {X 0,Y 93.515,Z 862.759,A -85,B 0,C 180,E1 -28088.644,E2 -28088.644} C_VEL
LIN {X 0,Y 101.389,Z 864.204,A -85,B 0,C 180,E1 -28093.962,E2 -28093.962} C_VEL
LIN {X 0,Y 111.578,Z 864.63,A -85,B 0,C 180,E1 -28099.122,E2 -28099.122} C_VEL
LIN {X 0,Y 123.056,Z 863.716,A -85,B 0,C 180,E1 -28103.564,E2 -28103.564} C_VEL
LIN {X 0,Y 124.235,Z 863.928,A -85,B 0,C 180,E1 -28105.159,E2 -28105.159} C_VEL
LIN {X 0,Y 119.242,Z 865.923,A -85,B 0,C 180,E1 -28107.86,E2 -28107.86} C_VEL
LIN {X 0,Y 108.362,Z 869.124,A -85,B 0,C 180,E1 -28112.526,E2 -28112.526} C_VEL
LIN {X 0,Y 98.128,Z 871.27,A -85,B 0,C 180,E1 -28118.016,E2 -28118.016} C_VEL
LIN {X 0,Y 88.908,Z 872.31,A -85,B 0,C 180,E1 -28124.647,E2 -28124.647} C_VEL
LIN {X 0,Y 81.284,Z 872.239,A -85,B 0,C 180,E1 -28132.753,E2 -28132.753} C_VEL
LIN {X 0,Y 76.232,Z 871.186,A -85,B 0,C 180,E1 -28142.55,E2 -28142.55} C_VEL
LIN {X 0,Y 74.022,Z 868.988,A -85,B 0,C 180,E1 -28153.45,E2 -28153.45} C_VEL
LIN {X 0,Y 74.788,Z 865.515,A -85,B 0,C 180,E1 -28164.607,E2 -28164.607} C_VEL
LIN {X 0,Y 75.33,Z 864.371,A -85,B 0,C 180,E1 -28167.326,E2 -28167.326} C_VEL
LIN {X 0,Y 75.105,Z 862.789,A -85,B 0,C 180,E1 -28169.999,E2 -28169.999} C_VEL
LIN {X 0,Y 74.238,Z 856.785,A -85,B 0,C 180,E1 -28178.163,E2 -28178.163} C_VEL
LIN {X 0,Y 74.778,Z 849.28,A -85,B 0,C 180,E1 -28186.376,E2 -28186.376} C_VEL
LIN {X 0,Y 75.262,Z 845.006,A -85,B 0,C 180,E1 -28190.232,E2 -28190.232} C_VEL
LIN {X 0,Y 75.251,Z 836.865,A -85,B 0,C 180,E1 -28196.335,E2 -28196.335} C_VEL
LIN {X 0,Y 75.68,Z 826.193,A -85,B 0,C 180,E1 -28202.908,E2 -28202.908} C_VEL
LIN {X 0,Y 76.552,Z 813.587,A -85,B 0,C 180,E1 -28209.136,E2 -28209.136} C_VEL
LIN {X 0,Y 77.582,Z 800.398,A -85,B 0,C 180,E1 -28214.164,E2 -28214.164} C_VEL
LIN {X 0,Y 78.466,Z 788.07,A -85,B 0,C 180,E1 -28217.795,E2 -28217.795} C_VEL
LIN {X 0,Y 74.857,Z 775.504,A -85,B 0,C 180,E1 -28222.081,E2 -28222.081} C_VEL
LIN {X 0,Y 73.735,Z 771.597,A -85,B 0,C 180,E1 -28223.437,E2 -28223.437} C_VEL
LIN {X 0,Y 72.781,Z 767.737,A -85,B 0,C 180,E1 -28231.131,E2 -28231.131} C_VEL
LIN {X 0,Y 72.673,Z 767.423,A -85,B 0,C 180,E1 -28232.655,E2 -28232.655} C_VEL
LIN {X 0,Y 72.722,Z 767.426,A -85,B 0,C 180,E1 -28245.109,E2 -28245.109} C_VEL
LIN {X 0,Y 72.858,Z 767.404,A -85,B 0,C 180,E1 -28248.877,E2 -28248.877} C_VEL
LIN {X 0,Y 73.559,Z 767.315,A -85,B 0,C 180,E1 -28260.001,E2 -28260.001} C_VEL
LIN {X 0,Y 72.831,Z 767.413,A -85,B 0,C 180,E1 -28271.128,E2 -28271.128} C_VEL
LIN {X 0,Y 72.508,Z 767.444,A -85,B 0,C 180,E1 -28276.906,E2 -28276.906} C_VEL
LIN {X 0,Y 72.37,Z 767.466,A -85,B 0,C 180,E1 -28282.859,E2 -28282.859} C_VEL
LIN {X 0,Y 72.358,Z 767.472,A -85,B 0,C 180,E1 -28289.055,E2 -28289.055} C_VEL
LIN {X 0,Y 72.289,Z 767.476,A -85,B 0,C 180,E1 -28295.686,E2 -28295.686} C_VEL
LIN {X 0,Y 72.242,Z 767.478,A -85,B 0,C 180,E1 -28302.922,E2 -28302.922} C_VEL
LIN {X 0,Y 72.291,Z 767.471,A -85,B 0,C 180,E1 -28311.056,E2 -28311.056} C_VEL
LIN {X 0,Y 72.282,Z 767.481,A -85,B 0,C 180,E1 -28314.312,E2 -28314.312} C_VEL
LIN {X 0,Y 72.314,Z 767.47,A -85,B 0,C 180,E1 -28321.009,E2 -28321.009} C_VEL
LIN {X 0,Y 72.345,Z 767.466,A -85,B 0,C 180,E1 -28327.134,E2 -28327.134} C_VEL
LIN {X 0,Y 72.678,Z 767.427,A -85,B 0,C 180,E1 -28335.244,E2 -28335.244} C_VEL
LIN {X 0,Y 72.826,Z 767.409,A -85,B 0,C 180,E1 -28338.872,E2 -28338.872} C_VEL
LIN {X 0,Y 73.545,Z 767.324,A -85,B 0,C 180,E1 -28350.001,E2 -28350.001} C_VEL
LIN {X 0,Y 72.86,Z 767.404,A -85,B 0,C 180,E1 -28361.124,E2 -28361.124} C_VEL
LIN {X 0,Y 72.812,Z 767.566,A -85,B 0,C 180,E1 -28363.225,E2 -28363.225} C_VEL
LIN {X 0,Y 76.764,Z 779.157,A -85,B 0,C 180,E1 -28368.687,E2 -28368.687} C_VEL
LIN {X 0,Y 79.807,Z 790.021,A -85,B 0,C 180,E1 -28374.035,E2 -28374.035} C_VEL
LIN {X 0,Y 80.273,Z 791.879,A -85,B 0,C 180,E1 -28374.981,E2 -28374.981} C_VEL
LIN {X 0,Y 80.245,Z 794.632,A -85,B 0,C 180,E1 -28376.236,E2 -28376.236} C_VEL
LIN {X 0,Y 78.77,Z 798.497,A -85,B 0,C 180,E1 -28377.748,E2 -28377.748} C_VEL
LIN {X 0,Y 73.057,Z 807.426,A -85,B 0,C 180,E1 -28381.535,E2 -28381.535} C_VEL
LIN {X 0,Y 72.398,Z 809.017,A -85,B 0,C 180,E1 -28382.424,E2 -28382.424} C_VEL
LIN {X 0,Y 69.344,Z 819.399,A -85,B 0,C 180,E1 -28389.394,E2 -28389.394} C_VEL
LIN {X 0,Y 66.854,Z 830.106,A -85,B 0,C 180,E1 -28398.879,E2 -28398.879} C_VEL
LIN {X 0,Y 65.884,Z 838.718,A -85,B 0,C 180,E1 -28408.582,E2 -28408.582} C_VEL
LIN {X 0,Y 66.64,Z 845.483,A -85,B 0,C 180,E1 -28417.896,E2 -28417.896} C_VEL
LIN {X 0,Y 69.576,Z 851.984,A -85,B 0,C 180,E1 -28428.344,E2 -28428.344} C_VEL
LIN {X 0,Y 74.313,Z 856.946,A -85,B 0,C 180,E1 -28437.289,E2 -28437.289} C_VEL
LIN {X 0,Y 80.567,Z 860.731,A -85,B 0,C 180,E1 -28445.004,E2 -28445.004} C_VEL
LIN {X 0,Y 85.5,Z 862.69,A -85,B 0,C 180,E1 -28449.462,E2 -28449.462} C_VEL
LIN {X 0,Y 95.082,Z 864.997,A -85,B 0,C 180,E1 -28456.073,E2 -28456.073} C_VEL
LIN {X 0,Y 105.592,Z 865.943,A -85,B 0,C 180,E1 -28461.278,E2 -28461.278} C_VEL
LIN {X 0,Y 114.095,Z 865.824,A -85,B 0,C 180,E1 -28464.568,E2 -28464.568} C_VEL
LIN {X 0,Y 113.416,Z 866.284,A -85,B 0,C 180,E1 -28465.707,E2 -28465.707} C_VEL
LIN {X 0,Y 104.692,Z 868.38,A -85,B 0,C 180,E1 -28469.225,E2 -28469.225} C_VEL
LIN {X 0,Y 93.916,Z 870.204,A -85,B 0,C 180,E1 -28474.596,E2 -28474.596} C_VEL
LIN {X 0,Y 84.107,Z 870.932,A -85,B 0,C 180,E1 -28481.231,E2 -28481.231} C_VEL
LIN {X 0,Y 75.843,Z 870.59,A -85,B 0,C 180,E1 -28489.559,E2 -28489.559} C_VEL
LIN {X 0,Y 70.153,Z 869.251,A -85,B 0,C 180,E1 -28499.939,E2 -28499.939} C_VEL
LIN {X 0,Y 67.485,Z 866.81,A -85,B 0,C 180,E1 -28511.794,E2 -28511.794} C_VEL
LIN {X 0,Y 68.094,Z 863.118,A -85,B 0,C 180,E1 -28524.075,E2 -28524.075} C_VEL
LIN {X 0,Y 68.568,Z 861.919,A -85,B 0,C 180,E1 -28527.062,E2 -28527.062} C_VEL
LIN {X 0,Y 67.637,Z 857.243,A -85,B 0,C 180,E1 -28534.469,E2 -28534.469} C_VEL
LIN {X 0,Y 67.556,Z 850.065,A -85,B 0,C 180,E1 -28543.536,E2 -28543.536} C_VEL
LIN {X 0,Y 68.208,Z 844.833,A -85,B 0,C 180,E1 -28549.024,E2 -28549.024} C_VEL
LIN {X 0,Y 68.228,Z 838.693,A -85,B 0,C 180,E1 -28554.332,E2 -28554.332} C_VEL
LIN {X 0,Y 68.528,Z 827.63,A -85,B 0,C 180,E1 -28562.315,E2 -28562.315} C_VEL
LIN {X 0,Y 69.378,Z 815.42,A -85,B 0,C 180,E1 -28569.28,E2 -28569.28} C_VEL
LIN {X 0,Y 70.625,Z 802.743,A -85,B 0,C 180,E1 -28574.937,E2 -28574.937} C_VEL
LIN {X 0,Y 71.782,Z 789.54,A -85,B 0,C 180,E1 -28579.409,E2 -28579.409} C_VEL
LIN {X 0,Y 68.762,Z 778.463,A -85,B 0,C 180,E1 -28583.781,E2 -28583.781} C_VEL
LIN {X 0,Y 66.214,Z 770.394,A -85,B 0,C 180,E1 -28587.046,E2 -28587.046} C_VEL
LIN {X 0,Y 65.656,Z 768.298,A -85,B 0,C 180,E1 -28592.076,E2 -28592.076} C_VEL
LIN {X 0,Y 65.626,Z 768.308,A -85,B 0,C 180,E1 -28604.541,E2 -28604.541} C_VEL
LIN {X 0,Y 65.755,Z 768.292,A -85,B 0,C 180,E1 -28607.658,E2 -28607.658} C_VEL
LIN {X 0,Y 66.483,Z 768.196,A -85,B 0,C 180,E1 -28620.001,E2 -28620.001} C_VEL
LIN {X 0,Y 65.723,Z 768.298,A -85,B 0,C 180,E1 -28632.35,E2 -28632.35} C_VEL
LIN {X 0,Y 65.338,Z 768.343,A -85,B 0,C 180,E1 -28638.826,E2 -28638.826} C_VEL
LIN {X 0,Y 65.216,Z 768.352,A -85,B 0,C 180,E1 -28645.536,E2 -28645.536} C_VEL
LIN {X 0,Y 65.168,Z 768.36,A -85,B 0,C 180,E1 -28652.632,E2 -28652.632} C_VEL
LIN {X 0,Y 65.178,Z 768.359,A -85,B 0,C 180,E1 -28660.993,E2 -28660.993} C_VEL
LIN {X 0,Y 65.198,Z 768.356,A -85,B 0,C 180,E1 -28669.702,E2 -28669.702} C_VEL
LIN {X 0,Y 65.196,Z 768.354,A -85,B 0,C 180,E1 -28679.588,E2 -28679.588} C_VEL
LIN {X 0,Y 65.187,Z 768.365,A -85,B 0,C 180,E1 -28684.454,E2 -28684.454} C_VEL
LIN {X 0,Y 65.58,Z 768.313,A -85,B 0,C 180,E1 -28694.69,E2 -28694.69} C_VEL
LIN {X 0,Y 65.72,Z 768.29,A -85,B 0,C 180,E1 -28697.651,E2 -28697.651} C_VEL
LIN {X 0,Y 66.443,Z 768.209,A -85,B 0,C 180,E1 -28710.001,E2 -28710.001} C_VEL
LIN {X 0,Y 65.812,Z 768.339,A -85,B 0,C 180,E1 -28720.188,E2 -28720.188} C_VEL
LIN {X 0,Y 69.652,Z 779.438,A -85,B 0,C 180,E1 -28726.225,E2 -28726.225} C_VEL
LIN {X 0,Y 72.531,Z 789.697,A -85,B 0,C 180,E1 -28731.772,E2 -28731.772} C_VEL
LIN {X 0,Y 74.756,Z 799.445,A -85,B 0,C 180,E1 -28737.279,E2 -28737.279} C_VEL
LIN {X 0,Y 74.944,Z 800.652,A -85,B 0,C 180,E1 -28737.962,E2 -28737.962} C_VEL
LIN {X 0,Y 72.398,Z 809.017,A -85,B 0,C 180,E1 -28742.424,E2 -28742.424} C_VEL
LIN {X 0,Y 70.354,Z 813.497,A -85,B 0,C 180,E1 -28745.051,E2 -28745.051} C_VEL
LIN {X 0,Y 65.554,Z 820.299,A -85,B 0,C 180,E1 -28749.605,E2 -28749.605} C_VEL
LIN {X 0,Y 61.075,Z 826.67,A -85,B 0,C 180,E1 -28755.227,E2 -28755.227} C_VEL
LIN {X 0,Y 59.638,Z 830.481,A -85,B 0,C 180,E1 -28759.331,E2 -28759.331} C_VEL
LIN {X 0,Y 58.831,Z 838.263,A -85,B 0,C 180,E1 -28769.056,E2 -28769.056} C_VEL
LIN {X 0,Y 60.227,Z 846.725,A -85,B 0,C 180,E1 -28781.726,E2 -28781.726} C_VEL
LIN {X 0,Y 64.421,Z 853.652,A -85,B 0,C 180,E1 -28793.736,E2 -28793.736} C_VEL
LIN {X 0,Y 70.384,Z 858.604,A -85,B 0,C 180,E1 -28803.098,E2 -28803.098} C_VEL
LIN {X 0,Y 78.947,Z 862.809,A -85,B 0,C 180,E1 -28811.69,E2 -28811.69} C_VEL
LIN {X 0,Y 88.929,Z 865.592,A -85,B 0,C 180,E1 -28818.492,E2 -28818.492} C_VEL
LIN {X 0,Y 99.805,Z 867.052,A -85,B 0,C 180,E1 -28823.732,E2 -28823.732} C_VEL
LIN {X 0,Y 101.702,Z 867.194,A -85,B 0,C 180,E1 -28824.495,E2 -28824.495} C_VEL
LIN {X 0,Y 101.391,Z 867.562,A -85,B 0,C 180,E1 -28825.695,E2 -28825.695} C_VEL
LIN {X 0,Y 90.071,Z 869.06,A -85,B 0,C 180,E1 -28830.872,E2 -28830.872} C_VEL
LIN {X 0,Y 79.647,Z 869.498,A -85,B 0,C 180,E1 -28837.423,E2 -28837.423} C_VEL
LIN {X 0,Y 70.696,Z 868.871,A -85,B 0,C 180,E1 -28845.901,E2 -28845.901} C_VEL
LIN {X 0,Y 64.247,Z 867.261,A -85,B 0,C 180,E1 -28856.841,E2 -28856.841} C_VEL
LIN {X 0,Y 61.034,Z 864.579,A -85,B 0,C 180,E1 -28869.79,E2 -28869.79} C_VEL
LIN {X 0,Y 61.438,Z 860.603,A -85,B 0,C 180,E1 -28883.431,E2 -28883.431} C_VEL
LIN {X 0,Y 61.795,Z 859.293,A -85,B 0,C 180,E1 -28886.739,E2 -28886.739} C_VEL
LIN {X 0,Y 60.618,Z 853.133,A -85,B 0,C 180,E1 -28896.657,E2 -28896.657} C_VEL
LIN {X 0,Y 61.081,Z 845.341,A -85,B 0,C 180,E1 -28906.717,E2 -28906.717} C_VEL
LIN {X 0,Y 61.245,Z 840.587,A -85,B 0,C 180,E1 -28911.647,E2 -28911.647} C_VEL
LIN {X 0,Y 61.273,Z 830.801,A -85,B 0,C 180,E1 -28920.119,E2 -28920.119} C_VEL
LIN {X 0,Y 61.971,Z 820.324,A -85,B 0,C 180,E1 -28927.453,E2 -28927.453} C_VEL
LIN {X 0,Y 63.219,Z 808.569,A -85,B 0,C 180,E1 -28934.011,E2 -28934.011} C_VEL
LIN {X 0,Y 64.653,Z 795.724,A -85,B 0,C 180,E1 -28939.545,E2 -28939.545} C_VEL
LIN {X 0,Y 64.972,Z 790.309,A -85,B 0,C 180,E1 -28941.536,E2 -28941.536} C_VEL
LIN {X 0,Y 61.651,Z 777.982,A -85,B 0,C 180,E1 -28947.212,E2 -28947.212} C_VEL
LIN {X 0,Y 59.717,Z 772.712,A -85,B 0,C 180,E1 -28949.901,E2 -28949.901} C_VEL
LIN {X 0,Y 58.617,Z 769.175,A -85,B 0,C 180,E1 -28951.708,E2 -28951.708} C_VEL
LIN {X 0,Y 58.633,Z 769.182,A -85,B 0,C 180,E1 -28966.13,E2 -28966.13} C_VEL
LIN {X 0,Y 58.799,Z 769.158,A -85,B 0,C 180,E1 -28973.136,E2 -28973.136} C_VEL
LIN {X 0,Y 59.373,Z 769.081,A -85,B 0,C 180,E1 -28980.001,E2 -28980.001} C_VEL
LIN {X 0,Y 58.783,Z 769.154,A -85,B 0,C 180,E1 -28986.867,E2 -28986.867} C_VEL
LIN {X 0,Y 58.457,Z 769.194,A -85,B 0,C 180,E1 -28995.888,E2 -28995.888} C_VEL
LIN {X 0,Y 58.158,Z 769.24,A -85,B 0,C 180,E1 -29001.256,E2 -29001.256} C_VEL
LIN {X 0,Y 58.125,Z 769.245,A -85,B 0,C 180,E1 -29008.925,E2 -29008.925} C_VEL
LIN {X 0,Y 58.02,Z 769.257,A -85,B 0,C 180,E1 -29017.277,E2 -29017.277} C_VEL
LIN {X 0,Y 58.008,Z 769.259,A -85,B 0,C 180,E1 -29026.631,E2 -29026.631} C_VEL
LIN {X 0,Y 58.014,Z 769.252,A -85,B 0,C 180,E1 -29032.72,E2 -29032.72} C_VEL
LIN {X 0,Y 58.1,Z 769.24,A -85,B 0,C 180,E1 -29041.063,E2 -29041.063} C_VEL
LIN {X 0,Y 58.143,Z 769.233,A -85,B 0,C 180,E1 -29048.739,E2 -29048.739} C_VEL
LIN {X 0,Y 58.592,Z 769.178,A -85,B 0,C 180,E1 -29056.12,E2 -29056.12} C_VEL
LIN {X 0,Y 58.77,Z 769.161,A -85,B 0,C 180,E1 -29063.133,E2 -29063.133} C_VEL
LIN {X 0,Y 59.336,Z 769.094,A -85,B 0,C 180,E1 -29070.001,E2 -29070.001} C_VEL
LIN {X 0,Y 58.829,Z 769.152,A -85,B 0,C 180,E1 -29076.431,E2 -29076.431} C_VEL
LIN {X 0,Y 62.112,Z 778.275,A -85,B 0,C 180,E1 -29082.25,E2 -29082.25} C_VEL
LIN {X 0,Y 64.603,Z 786.585,A -85,B 0,C 180,E1 -29087.408,E2 -29087.408} C_VEL
LIN {X 0,Y 66.876,Z 795.94,A -85,B 0,C 180,E1 -29093.21,E2 -29093.21} C_VEL
LIN {X 0,Y 67.818,Z 800.512,A -85,B 0,C 180,E1 -29096.132,E2 -29096.132} C_VEL
LIN {X 0,Y 67.028,Z 804.135,A -85,B 0,C 180,E1 -29098.154,E2 -29098.154} C_VEL
LIN {X 0,Y 63.414,Z 815.456,A -85,B 0,C 180,E1 -29105.459,E2 -29105.459} C_VEL
LIN {X 0,Y 60.632,Z 825.48,A -85,B 0,C 180,E1 -29114.066,E2 -29114.066} C_VEL
LIN {X 0,Y 59.638,Z 830.481,A -85,B 0,C 180,E1 -29119.331,E2 -29119.331} C_VEL
LIN {X 0,Y 58.439,Z 834.14,A -85,B 0,C 180,E1 -29123.683,E2 -29123.683} C_VEL
LIN {X 0,Y 55.374,Z 839.57,A -85,B 0,C 180,E1 -29131.457,E2 -29131.457} C_VEL
LIN {X 0,Y 53.397,Z 844.569,A -85,B 0,C 180,E1 -29140.307,E2 -29140.307} C_VEL
LIN {X 0,Y 53.906,Z 847.522,A -85,B 0,C 180,E1 -29145.775,E2 -29145.775} C_VEL
LIN {X 0,Y 58.139,Z 853.563,A -85,B 0,C 180,E1 -29156.843,E2 -29156.843} C_VEL
LIN {X 0,Y 64.336,Z 858.556,A -85,B 0,C 180,E1 -29166.271,E2 -29166.271} C_VEL
LIN {X 0,Y 72.549,Z 862.706,A -85,B 0,C 180,E1 -29174.365,E2 -29174.365} C_VEL
LIN {X 0,Y 82.971,Z 865.987,A -85,B 0,C 180,E1 -29181.289,E2 -29181.289} C_VEL
LIN {X 0,Y 89.509,Z 867.307,A -85,B 0,C 180,E1 -29184.513,E2 -29184.513} C_VEL
LIN {X 0,Y 86.651,Z 867.77,A -85,B 0,C 180,E1 -29186.85,E2 -29186.85} C_VEL
LIN {X 0,Y 75.605,Z 867.911,A -85,B 0,C 180,E1 -29193.214,E2 -29193.214} C_VEL
LIN {X 0,Y 65.909,Z 867.005,A -85,B 0,C 180,E1 -29201.717,E2 -29201.717} C_VEL
LIN {X 0,Y 58.621,Z 865.138,A -85,B 0,C 180,E1 -29213.169,E2 -29213.169} C_VEL
LIN {X 0,Y 54.723,Z 862.179,A -85,B 0,C 180,E1 -29227.337,E2 -29227.337} C_VEL
LIN {X 0,Y 54.817,Z 858.026,A -85,B 0,C 180,E1 -29242.633,E2 -29242.633} C_VEL
LIN {X 0,Y 54.973,Z 856.511,A -85,B 0,C 180,E1 -29246.334,E2 -29246.334} C_VEL
LIN {X 0,Y 53.884,Z 851.153,A -85,B 0,C 180,E1 -29255.613,E2 -29255.613} C_VEL
LIN {X 0,Y 54.219,Z 843.167,A -85,B 0,C 180,E1 -29266.956,E2 -29266.956} C_VEL
LIN {X 0,Y 54.132,Z 837.865,A -85,B 0,C 180,E1 -29272.922,E2 -29272.922} C_VEL
LIN {X 0,Y 54.347,Z 827.95,A -85,B 0,C 180,E1 -29282.237,E2 -29282.237} C_VEL
LIN {X 0,Y 55.265,Z 816.81,A -85,B 0,C 180,E1 -29290.693,E2 -29290.693} C_VEL
LIN {X 0,Y 56.857,Z 804.604,A -85,B 0,C 180,E1 -29297.871,E2 -29297.871} C_VEL
LIN {X 0,Y 58.335,Z 793.357,A -85,B 0,C 180,E1 -29302.96,E2 -29302.96} C_VEL
LIN {X 0,Y 57.758,Z 789.214,A -85,B 0,C 180,E1 -29305.069,E2 -29305.069} C_VEL
LIN {X 0,Y 54.718,Z 777.721,A -85,B 0,C 180,E1 -29311.469,E2 -29311.469} C_VEL
LIN {X 0,Y 52.957,Z 773.628,A -85,B 0,C 180,E1 -29314.186,E2 -29314.186} C_VEL
LIN {X 0,Y 51.579,Z 771.171,A -85,B 0,C 180,E1 -29316.139,E2 -29316.139} C_VEL
LIN {X 0,Y 51.338,Z 770.09,A -85,B 0,C 180,E1 -29316.817,E2 -29316.817} C_VEL
LIN {X 0,Y 51.471,Z 770.07,A -85,B 0,C 180,E1 -29324.153,E2 -29324.153} C_VEL
LIN {X 0,Y 51.676,Z 770.041,A -85,B 0,C 180,E1 -29332.184,E2 -29332.184} C_VEL
LIN {X 0,Y 52.255,Z 769.967,A -85,B 0,C 180,E1 -29340.001,E2 -29340.001} C_VEL
LIN {X 0,Y 51.656,Z 770.04,A -85,B 0,C 180,E1 -29347.82,E2 -29347.82} C_VEL
LIN {X 0,Y 51.336,Z 770.08,A -85,B 0,C 180,E1 -29356.603,E2 -29356.603} C_VEL
LIN {X 0,Y 50.998,Z 770.123,A -85,B 0,C 180,E1 -29364.421,E2 -29364.421} C_VEL
LIN {X 0,Y 50.985,Z 770.125,A -85,B 0,C 180,E1 -29374.202,E2 -29374.202} C_VEL
LIN {X 0,Y 50.975,Z 770.127,A -85,B 0,C 180,E1 -29383.581,E2 -29383.581} C_VEL
LIN {X 0,Y 50.975,Z 770.136,A -85,B 0,C 180,E1 -29386.422,E2 -29386.422} C_VEL
LIN {X 0,Y 50.995,Z 770.132,A -85,B 0,C 180,E1 -29396.547,E2 -29396.547} C_VEL
LIN {X 0,Y 50.98,Z 770.132,A -85,B 0,C 180,E1 -29405.571,E2 -29405.571} C_VEL
LIN {X 0,Y 51.371,Z 770.084,A -85,B 0,C 180,E1 -29414.121,E2 -29414.121} C_VEL
LIN {X 0,Y 51.647,Z 770.051,A -85,B 0,C 180,E1 -29422.18,E2 -29422.18} C_VEL
LIN {X 0,Y 52.147,Z 769.988,A -85,B 0,C 180,E1 -29430.966,E2 -29430.966} C_VEL
LIN {X 0,Y 52.068,Z 770.068,A -85,B 0,C 180,E1 -29431.935,E2 -29431.935} C_VEL
LIN {X 0,Y 52.8,Z 772.664,A -85,B 0,C 180,E1 -29433.817,E2 -29433.817} C_VEL
LIN {X 0,Y 55.474,Z 779.467,A -85,B 0,C 180,E1 -29439.113,E2 -29439.113} C_VEL
LIN {X 0,Y 58.147,Z 789.008,A -85,B 0,C 180,E1 -29445.781,E2 -29445.781} C_VEL
LIN {X 0,Y 60.244,Z 798.237,A -85,B 0,C 180,E1 -29452.282,E2 -29452.282} C_VEL
LIN {X 0,Y 60.926,Z 801.885,A -85,B 0,C 180,E1 -29454.929,E2 -29454.929} C_VEL
LIN {X 0,Y 57.183,Z 813.146,A -85,B 0,C 180,E1 -29462.331,E2 -29462.331} C_VEL
LIN {X 0,Y 53.921,Z 823.767,A -85,B 0,C 180,E1 -29471.959,E2 -29471.959} C_VEL
LIN {X 0,Y 52.087,Z 833.329,A -85,B 0,C 180,E1 -29483.344,E2 -29483.344} C_VEL
LIN {X 0,Y 52.132,Z 841.9,A -85,B 0,C 180,E1 -29496.143,E2 -29496.143} C_VEL
LIN {X 0,Y 53.906,Z 847.522,A -85,B 0,C 180,E1 -29505.775,E2 -29505.775} C_VEL
LIN {X 0,Y 54.904,Z 850.352,A -85,B 0,C 180,E1 -29511.14,E2 -29511.14} C_VEL
LIN {X 0,Y 56.035,Z 854.514,A -85,B 0,C 180,E1 -29520.38,E2 -29520.38} C_VEL
LIN {X 0,Y 58.683,Z 858.172,A -85,B 0,C 180,E1 -29529.223,E2 -29529.223} C_VEL
LIN {X 0,Y 61.818,Z 860.212,A -85,B 0,C 180,E1 -29533.583,E2 -29533.583} C_VEL
LIN {X 0,Y 73.54,Z 865.092,A -85,B 0,C 180,E1 -29542.474,E2 -29542.474} C_VEL
LIN {X 0,Y 77.264,Z 866.186,A -85,B 0,C 180,E1 -29544.546,E2 -29544.546} C_VEL
LIN {X 0,Y 77.761,Z 866.455,A -85,B 0,C 180,E1 -29545.337,E2 -29545.337} C_VEL
LIN {X 0,Y 66.56,Z 865.766,A -85,B 0,C 180,E1 -29552.357,E2 -29552.357} C_VEL
LIN {X 0,Y 57.05,Z 864.096,A -85,B 0,C 180,E1 -29562.341,E2 -29562.341} C_VEL
LIN {X 0,Y 50.055,Z 861.185,A -85,B 0,C 180,E1 -29577.398,E2 -29577.398} C_VEL
LIN {X 0,Y 47.866,Z 857.646,A -85,B 0,C 180,E1 -29592.922,E2 -29592.922} C_VEL
LIN {X 0,Y 48.29,Z 855.258,A -85,B 0,C 180,E1 -29601.631,E2 -29601.631} C_VEL
LIN {X 0,Y 48.181,Z 853.621,A -85,B 0,C 180,E1 -29605.817,E2 -29605.817} C_VEL
LIN {X 0,Y 46.992,Z 846.648,A -85,B 0,C 180,E1 -29618.6,E2 -29618.6} C_VEL
LIN {X 0,Y 47.308,Z 840.967,A -85,B 0,C 180,E1 -29627.284,E2 -29627.284} C_VEL
LIN {X 0,Y 46.987,Z 833.214,A -85,B 0,C 180,E1 -29636.661,E2 -29636.661} C_VEL
LIN {X 0,Y 47.523,Z 823.716,A -85,B 0,C 180,E1 -29646.266,E2 -29646.266} C_VEL
LIN {X 0,Y 49.067,Z 811.819,A -85,B 0,C 180,E1 -29655.738,E2 -29655.738} C_VEL
LIN {X 0,Y 50.928,Z 799.877,A -85,B 0,C 180,E1 -29663.005,E2 -29663.005} C_VEL
LIN {X 0,Y 51.808,Z 793.787,A -85,B 0,C 180,E1 -29665.988,E2 -29665.988} C_VEL
LIN {X 0,Y 49.936,Z 784.873,A -85,B 0,C 180,E1 -29671.641,E2 -29671.641} C_VEL
LIN {X 0,Y 48.003,Z 778.402,A -85,B 0,C 180,E1 -29676.259,E2 -29676.259} C_VEL
LIN {X 0,Y 45.723,Z 774.441,A -85,B 0,C 180,E1 -29680.329,E2 -29680.329} C_VEL
LIN {X 0,Y 44.521,Z 771.76,A -85,B 0,C 180,E1 -29683.024,E2 -29683.024} C_VEL
LIN {X 0,Y 44.397,Z 770.948,A -85,B 0,C 180,E1 -29683.761,E2 -29683.761} C_VEL
LIN {X 0,Y 44.532,Z 770.928,A -85,B 0,C 180,E1 -29690.921,E2 -29690.921} C_VEL
LIN {X 0,Y 45.128,Z 770.854,A -85,B 0,C 180,E1 -29700.001,E2 -29700.001} C_VEL
LIN {X 0,Y 44.499,Z 770.933,A -85,B 0,C 180,E1 -29709.088,E2 -29709.088} C_VEL
LIN {X 0,Y 44.105,Z 770.985,A -85,B 0,C 180,E1 -29718.585,E2 -29718.585} C_VEL
LIN {X 0,Y 43.813,Z 771.027,A -85,B 0,C 180,E1 -29728.767,E2 -29728.767} C_VEL
LIN {X 0,Y 43.784,Z 771.026,A -85,B 0,C 180,E1 -29739.948,E2 -29739.948} C_VEL
LIN {X 0,Y 43.819,Z 771.021,A -85,B 0,C 180,E1 -29753.318,E2 -29753.318} C_VEL
LIN {X 0,Y 43.797,Z 771.021,A -85,B 0,C 180,E1 -29761.224,E2 -29761.224} C_VEL
LIN {X 0,Y 44.169,Z 770.984,A -85,B 0,C 180,E1 -29772.693,E2 -29772.693} C_VEL
LIN {X 0,Y 44.706,Z 770.906,A -85,B 0,C 180,E1 -29784.928,E2 -29784.928} C_VEL
LIN {X 0,Y 45.776,Z 773.535,A -85,B 0,C 180,E1 -29787.801,E2 -29787.801} C_VEL
LIN {X 0,Y 47.355,Z 776.56,A -85,B 0,C 180,E1 -29791.17,E2 -29791.17} C_VEL
LIN {X 0,Y 49.571,Z 782.925,A -85,B 0,C 180,E1 -29797.045,E2 -29797.045} C_VEL
LIN {X 0,Y 51.884,Z 792.343,A -85,B 0,C 180,E1 -29804.714,E2 -29804.714} C_VEL
LIN {X 0,Y 53.753,Z 801.443,A -85,B 0,C 180,E1 -29812.081,E2 -29812.081} C_VEL
LIN {X 0,Y 53.965,Z 802.554,A -85,B 0,C 180,E1 -29812.999,E2 -29812.999} C_VEL
LIN {X 0,Y 50.123,Z 813.25,A -85,B 0,C 180,E1 -29820.814,E2 -29820.814} C_VEL
LIN {X 0,Y 46.801,Z 823.685,A -85,B 0,C 180,E1 -29831.336,E2 -29831.336} C_VEL
LIN {X 0,Y 44.956,Z 833.171,A -85,B 0,C 180,E1 -29844.108,E2 -29844.108} C_VEL
LIN {X 0,Y 45.31,Z 841.718,A -85,B 0,C 180,E1 -29858.541,E2 -29858.541} C_VEL
LIN {X 0,Y 48.217,Z 848.653,A -85,B 0,C 180,E1 -29871.618,E2 -29871.618} C_VEL
LIN {X 0,Y 53.896,Z 854.984,A -85,B 0,C 180,E1 -29883.738,E2 -29883.738} C_VEL
LIN {X 0,Y 61.818,Z 860.212,A -85,B 0,C 180,E1 -29893.583,E2 -29893.583} C_VEL
LIN {X 0,Y 62.808,Z 861.001,A -85,B 0,C 180,E1 -29895.534,E2 -29895.534} C_VEL
LIN {X 0,Y 62.753,Z 861.808,A -85,B 0,C 180,E1 -29898.579,E2 -29898.579} C_VEL
LIN {X 0,Y 61.321,Z 862.414,A -85,B 0,C 180,E1 -29902.659,E2 -29902.659} C_VEL
LIN {X 0,Y 59.533,Z 862.56,A -85,B 0,C 180,E1 -29905.857,E2 -29905.857} C_VEL
LIN {X 0,Y 55.667,Z 862.338,A -85,B 0,C 180,E1 -29911.704,E2 -29911.704} C_VEL
LIN {X 0,Y 50.398,Z 861.246,A -85,B 0,C 180,E1 -29920.032,E2 -29920.032} C_VEL
LIN {X 0,Y 49.096,Z 860.811,A -85,B 0,C 180,E1 -29922.239,E2 -29922.239} C_VEL
LIN {X 0,Y 42.664,Z 857.13,A -85,B 0,C 180,E1 -29940.383,E2 -29940.383} C_VEL
LIN {X 0,Y 41.834,Z 852.415,A -85,B 0,C 180,E1 -29960.327,E2 -29960.327} C_VEL
LIN {X 0,Y 41.073,Z 849.412,A -85,B 0,C 180,E1 -29967.547,E2 -29967.547} C_VEL
LIN {X 0,Y 40.319,Z 841.673,A -85,B 0,C 180,E1 -29982.584,E2 -29982.584} C_VEL
LIN {X 0,Y 40.315,Z 838.487,A -85,B 0,C 180,E1 -29987.762,E2 -29987.762} C_VEL
LIN {X 0,Y 40.153,Z 828.149,A -85,B 0,C 180,E1 -30001.674,E2 -30001.674} C_VEL
LIN {X 0,Y 41.224,Z 817.552,A -85,B 0,C 180,E1 -30012.994,E2 -30012.994} C_VEL
LIN {X 0,Y 43.393,Z 805.184,A -85,B 0,C 180,E1 -30022.96,E2 -30022.96} C_VEL
LIN {X 0,Y 45.065,Z 796.526,A -85,B 0,C 180,E1 -30028.243,E2 -30028.243} C_VEL
LIN {X 0,Y 45.049,Z 793.646,A -85,B 0,C 180,E1 -30030.181,E2 -30030.181} C_VEL
LIN {X 0,Y 43.273,Z 784.649,A -85,B 0,C 180,E1 -30037.312,E2 -30037.312} C_VEL
LIN {X 0,Y 42.133,Z 781.514,A -85,B 0,C 180,E1 -30040.513,E2 -30040.513} C_VEL
LIN {X 0,Y 39.411,Z 775.986,A -85,B 0,C 180,E1 -30047.571,E2 -30047.571} C_VEL
LIN {X 0,Y 37.833,Z 773.214,A -85,B 0,C 180,E1 -30051.992,E2 -30051.992} C_VEL
LIN {X 0,Y 37.551,Z 771.806,A -85,B 0,C 180,E1 -30053.958,E2 -30053.958} C_VEL
LIN {X 0,Y 37.983,Z 771.744,A -85,B 0,C 180,E1 -30060.001,E2 -30060.001} C_VEL
LIN {X 0,Y 37.294,Z 771.836,A -85,B 0,C 180,E1 -30070.864,E2 -30070.864} C_VEL
LIN {X 0,Y 37.028,Z 771.865,A -85,B 0,C 180,E1 -30078.377,E2 -30078.377} C_VEL
LIN {X 0,Y 36.694,Z 771.905,A -85,B 0,C 180,E1 -30095.072,E2 -30095.072} C_VEL
LIN {X 0,Y 36.709,Z 771.906,A -85,B 0,C 180,E1 -30100.022,E2 -30100.022} C_VEL
LIN {X 0,Y 36.711,Z 771.902,A -85,B 0,C 180,E1 -30109.977,E2 -30109.977} C_VEL
LIN {X 0,Y 36.697,Z 771.914,A -85,B 0,C 180,E1 -30114.933,E2 -30114.933} C_VEL
LIN {X 0,Y 37.109,Z 771.863,A -85,B 0,C 180,E1 -30132.844,E2 -30132.844} C_VEL
LIN {X 0,Y 37.146,Z 772.084,A -85,B 0,C 180,E1 -30134.164,E2 -30134.164} C_VEL
LIN {X 0,Y 37.948,Z 774.236,A -85,B 0,C 180,E1 -30137.556,E2 -30137.556} C_VEL
LIN {X 0,Y 40.017,Z 776.435,A -85,B 0,C 180,E1 -30142.686,E2 -30142.686} C_VEL
LIN {X 0,Y 42.175,Z 781.181,A -85,B 0,C 180,E1 -30149.035,E2 -30149.035} C_VEL
LIN {X 0,Y 43.99,Z 787.688,A -85,B 0,C 180,E1 -30155.732,E2 -30155.732} C_VEL
LIN {X 0,Y 45.523,Z 795.064,A -85,B 0,C 180,E1 -30162.823,E2 -30162.823} C_VEL
LIN {X 0,Y 46.896,Z 802.49,A -85,B 0,C 180,E1 -30169.887,E2 -30169.887} C_VEL
LIN {X 0,Y 46.91,Z 803.535,A -85,B 0,C 180,E1 -30170.81,E2 -30170.81} C_VEL
LIN {X 0,Y 42.579,Z 814.852,A -85,B 0,C 180,E1 -30180.281,E2 -30180.281} C_VEL
LIN {X 0,Y 39.297,Z 824.922,A -85,B 0,C 180,E1 -30192.459,E2 -30192.459} C_VEL
LIN {X 0,Y 37.828,Z 833.38,A -85,B 0,C 180,E1 -30206.125,E2 -30206.125} C_VEL
LIN {X 0,Y 39.006,Z 842.666,A -85,B 0,C 180,E1 -30224.319,E2 -30224.319} C_VEL
LIN {X 0,Y 43.584,Z 850.269,A -85,B 0,C 180,E1 -30239.999,E2 -30239.999} C_VEL
LIN {X 0,Y 51.804,Z 857.146,A -85,B 0,C 180,E1 -30253.295,E2 -30253.295} C_VEL
LIN {X 0,Y 63.17,Z 863.09,A -85,B 0,C 180,E1 -30263.382,E2 -30263.382} C_VEL
LIN {X 0,Y 66.059,Z 864.188,A -85,B 0,C 180,E1 -30265.185,E2 -30265.185} C_VEL
LIN {X 0,Y 57.677,Z 863.004,A -85,B 0,C 180,E1 -30271.463,E2 -30271.463} C_VEL
LIN {X 0,Y 49.096,Z 860.811,A -85,B 0,C 180,E1 -30282.239,E2 -30282.239} C_VEL
LIN {X 0,Y 44.756,Z 858.932,A -85,B 0,C 180,E1 -30289.96,E2 -30289.96} C_VEL
LIN {X 0,Y 40.714,Z 856.296,A -85,B 0,C 180,E1 -30298.378,E2 -30298.378} C_VEL
LIN {X 0,Y 37.398,Z 853.064,A -85,B 0,C 180,E1 -30307.919,E2 -30307.919} C_VEL
LIN {X 0,Y 35.359,Z 849.391,A -85,B 0,C 180,E1 -30318.614,E2 -30318.614} C_VEL
LIN {X 0,Y 34.646,Z 847.28,A -85,B 0,C 180,E1 -30324.177,E2 -30324.177} C_VEL
LIN {X 0,Y 33.514,Z 839.342,A -85,B 0,C 180,E1 -30342.104,E2 -30342.104} C_VEL
LIN {X 0,Y 33.028,Z 833.898,A -85,B 0,C 180,E1 -30351.861,E2 -30351.861} C_VEL
LIN {X 0,Y 33.353,Z 824.029,A -85,B 0,C 180,E1 -30366.862,E2 -30366.862} C_VEL
LIN {X 0,Y 35.299,Z 812.39,A -85,B 0,C 180,E1 -30380.488,E2 -30380.488} C_VEL
LIN {X 0,Y 37.908,Z 800.598,A -85,B 0,C 180,E1 -30390.333,E2 -30390.333} C_VEL
LIN {X 0,Y 38.848,Z 796.422,A -85,B 0,C 180,E1 -30393.117,E2 -30393.117} C_VEL
LIN {X 0,Y 37.679,Z 788.019,A -85,B 0,C 180,E1 -30401.232,E2 -30401.232} C_VEL
LIN {X 0,Y 36.549,Z 784.644,A -85,B 0,C 180,E1 -30405.452,E2 -30405.452} C_VEL
LIN {X 0,Y 34.921,Z 780.997,A -85,B 0,C 180,E1 -30411.32,E2 -30411.32} C_VEL
LIN {X 0,Y 33.581,Z 777.983,A -85,B 0,C 180,E1 -30417.002,E2 -30417.002} C_VEL
LIN {X 0,Y 32.905,Z 776.797,A -85,B 0,C 180,E1 -30420.001,E2 -30420.001} C_VEL
LIN {X 0,Y 30.338,Z 773.941,A -85,B 0,C 180,E1 -30433.396,E2 -30433.396} C_VEL
LIN {X 0,Y 29.877,Z 772.637,A -85,B 0,C 180,E1 -30438.959,E2 -30438.959} C_VEL
LIN {X 0,Y 29.468,Z 772.676,A -85,B 0,C 180,E1 -30448.49,E2 -30448.49} C_VEL
LIN {X 0,Y 29.542,Z 772.712,A -85,B 0,C 180,E1 -30467.116,E2 -30467.116} C_VEL
LIN {X 0,Y 31.302,Z 776.666,A -85,B 0,C 180,E1 -30483.913,E2 -30483.913} C_VEL
LIN {X 0,Y 33.241,Z 778.312,A -85,B 0,C 180,E1 -30491.547,E2 -30491.547} C_VEL
LIN {X 0,Y 35.607,Z 782.142,A -85,B 0,C 180,E1 -30500.722,E2 -30500.722} C_VEL
LIN {X 0,Y 36.836,Z 785.384,A -85,B 0,C 180,E1 -30505.894,E2 -30505.894} C_VEL
LIN {X 0,Y 38.028,Z 790.822,A -85,B 0,C 180,E1 -30512.649,E2 -30512.649} C_VEL
LIN {X 0,Y 39.398,Z 799.211,A -85,B 0,C 180,E1 -30522.135,E2 -30522.135} C_VEL
LIN {X 0,Y 40.135,Z 804.056,A -85,B 0,C 180,E1 -30527.563,E2 -30527.563} C_VEL
LIN {X 0,Y 35.185,Z 815.87,A -85,B 0,C 180,E1 -30539.085,E2 -30539.085} C_VEL
LIN {X 0,Y 31.842,Z 826.039,A -85,B 0,C 180,E1 -30554.205,E2 -30554.205} C_VEL
LIN {X 0,Y 30.894,Z 836.407,A -85,B 0,C 180,E1 -30575.502,E2 -30575.502} C_VEL
LIN {X 0,Y 33.648,Z 844.307,A -85,B 0,C 180,E1 -30593.996,E2 -30593.996} C_VEL
LIN {X 0,Y 40.089,Z 851.76,A -85,B 0,C 180,E1 -30610.096,E2 -30610.096} C_VEL
LIN {X 0,Y 48.752,Z 857.896,A -85,B 0,C 180,E1 -30621.124,E2 -30621.124} C_VEL
LIN {X 0,Y 53.441,Z 860.415,A -85,B 0,C 180,E1 -30625.089,E2 -30625.089} C_VEL
LIN {X 0,Y 50.966,Z 860.063,A -85,B 0,C 180,E1 -30628.396,E2 -30628.396} C_VEL
LIN {X 0,Y 40.005,Z 856.388,A -85,B 0,C 180,E1 -30645.353,E2 -30645.353} C_VEL
LIN {X 0,Y 35.485,Z 852.074,A -85,B 0,C 180,E1 -30666.663,E2 -30666.663} C_VEL
LIN {X 0,Y 35.359,Z 849.391,A -85,B 0,C 180,E1 -30678.614,E2 -30678.614} C_VEL
LIN {X 0,Y 34.484,Z 847.317,A -85,B 0,C 180,E1 -30683.821,E2 -30683.821} C_VEL
LIN {X 0,Y 33.194,Z 844.971,A -85,B 0,C 180,E1 -30688.644,E2 -30688.644} C_VEL
LIN {X 0,Y 30.828,Z 841.099,A -85,B 0,C 180,E1 -30695.629,E2 -30695.629} C_VEL
LIN {X 0,Y 26.996,Z 834.008,A -85,B 0,C 180,E1 -30708.41,E2 -30708.41} C_VEL
LIN {X 0,Y 25.93,Z 829.466,A -85,B 0,C 180,E1 -30717.279,E2 -30717.279} C_VEL
LIN {X 0,Y 25.951,Z 827.892,A -85,B 0,C 180,E1 -30720.308,E2 -30720.308} C_VEL
LIN {X 0,Y 27.339,Z 817.42,A -85,B 0,C 180,E1 -30738.005,E2 -30738.005} C_VEL
LIN {X 0,Y 30.145,Z 806.612,A -85,B 0,C 180,E1 -30750.958,E2 -30750.958} C_VEL
LIN {X 0,Y 32.618,Z 797.63,A -85,B 0,C 180,E1 -30758.599,E2 -30758.599} C_VEL
LIN {X 0,Y 32.003,Z 790.414,A -85,B 0,C 180,E1 -30767.315,E2 -30767.315} C_VEL
LIN {X 0,Y 30.001,Z 784.798,A -85,B 0,C 180,E1 -30778.524,E2 -30778.524} C_VEL
LIN {X 0,Y 29.281,Z 782.717,A -85,B 0,C 180,E1 -30783.786,E2 -30783.786} C_VEL
LIN {X 0,Y 27.656,Z 780.613,A -85,B 0,C 180,E1 -30794.723,E2 -30794.723} C_VEL
LIN {X 0,Y 26.613,Z 779.253,A -85,B 0,C 180,E1 -30811.883,E2 -30811.883} C_VEL
LIN {X 0,Y 26.642,Z 779.259,A -85,B 0,C 180,E1 -30817.687,E2 -30817.687} C_VEL
LIN {X 0,Y 27.076,Z 780.756,A -85,B 0,C 180,E1 -30831.145,E2 -30831.145} C_VEL
LIN {X 0,Y 28.767,Z 783.607,A -85,B 0,C 180,E1 -30845.999,E2 -30845.999} C_VEL
LIN {X 0,Y 30.856,Z 786.981,A -85,B 0,C 180,E1 -30856.836,E2 -30856.836} C_VEL
LIN {X 0,Y 31.534,Z 789.027,A -85,B 0,C 180,E1 -30860.952,E2 -30860.952} C_VEL
LIN {X 0,Y 32.326,Z 795.027,A -85,B 0,C 180,E1 -30870.001,E2 -30870.001} C_VEL
LIN {X 0,Y 33.258,Z 803.869,A -85,B 0,C 180,E1 -30882.201,E2 -30882.201} C_VEL
LIN {X 0,Y 33.244,Z 804.914,A -85,B 0,C 180,E1 -30883.544,E2 -30883.544} C_VEL
LIN {X 0,Y 27.826,Z 816.803,A -85,B 0,C 180,E1 -30897.26,E2 -30897.26} C_VEL
LIN {X 0,Y 24.624,Z 826.058,A -85,B 0,C 180,E1 -30914.474,E2 -30914.474} C_VEL
LIN {X 0,Y 24.008,Z 835.026,A -85,B 0,C 180,E1 -30937.825,E2 -30937.825} C_VEL
LIN {X 0,Y 28.141,Z 844.066,A -85,B 0,C 180,E1 -30962.54,E2 -30962.54} C_VEL
LIN {X 0,Y 36.65,Z 852.209,A -85,B 0,C 180,E1 -30979.901,E2 -30979.901} C_VEL
LIN {X 0,Y 42.667,Z 856.211,A -85,B 0,C 180,E1 -30986.481,E2 -30986.481} C_VEL
LIN {X 0,Y 33.575,Z 852.645,A -85,B 0,C 180,E1 -31002.891,E2 -31002.891} C_VEL
LIN {X 0,Y 29.185,Z 847.749,A -85,B 0,C 180,E1 -31028.831,E2 -31028.831} C_VEL
LIN {X 0,Y 29.057,Z 846.209,A -85,B 0,C 180,E1 -31036.001,E2 -31036.001} C_VEL
LIN {X 0,Y 26.786,Z 838.422,A -85,B 0,C 180,E1 -31057.537,E2 -31057.537} C_VEL
LIN {X 0,Y 26.32,Z 835.026,A -85,B 0,C 180,E1 -31065.486,E2 -31065.486} C_VEL
LIN {X 0,Y 25.951,Z 827.892,A -85,B 0,C 180,E1 -31080.308,E2 -31080.308} C_VEL
LIN {X 0,Y 25.804,Z 823.382,A -85,B 0,C 180,E1 -31088.644,E2 -31088.644} C_VEL
LIN {X 0,Y 25.034,Z 818.758,A -85,B 0,C 180,E1 -31096.936,E2 -31096.936} C_VEL
LIN {X 0,Y 24.196,Z 807.612,A -85,B 0,C 180,E1 -31116.558,E2 -31116.558} C_VEL
LIN {X 0,Y 25.443,Z 802.456,A -85,B 0,C 180,E1 -31123.012,E2 -31123.012} C_VEL
LIN {X 0,Y 26.73,Z 798.518,A -85,B 0,C 180,E1 -31126.701,E2 -31126.701} C_VEL
LIN {X 0,Y 26.789,Z 794.752,A -85,B 0,C 180,E1 -31132.464,E2 -31132.464} C_VEL
LIN {X 0,Y 26.155,Z 791.356,A -85,B 0,C 180,E1 -31140.002,E2 -31140.002} C_VEL
LIN {X 0,Y 25.339,Z 788.286,A -85,B 0,C 180,E1 -31149.448,E2 -31149.448} C_VEL
LIN {X 0,Y 24.652,Z 787.087,A -85,B 0,C 180,E1 -31156.566,E2 -31156.566} C_VEL
LIN {X 0,Y 23.98,Z 785.836,A -85,B 0,C 180,E1 -31175.888,E2 -31175.888} C_VEL
LIN {X 0,Y 24.014,Z 786.873,A -85,B 0,C 180,E1 -31186.482,E2 -31186.482} C_VEL
LIN {X 0,Y 25.601,Z 790.738,A -85,B 0,C 180,E1 -31208.104,E2 -31208.104} C_VEL
LIN {X 0,Y 26.414,Z 793.295,A -85,B 0,C 180,E1 -31215.748,E2 -31215.748} C_VEL
LIN {X 0,Y 26.652,Z 799.473,A -85,B 0,C 180,E1 -31226.891,E2 -31226.891} C_VEL
LIN {X 0,Y 26.765,Z 804.577,A -85,B 0,C 180,E1 -31235.653,E2 -31235.653} C_VEL
LIN {X 0,Y 26.532,Z 805.905,A -85,B 0,C 180,E1 -31237.612,E2 -31237.612} C_VEL
LIN {X 0,Y 20.291,Z 818.091,A -85,B 0,C 180,E1 -31255.058,E2 -31255.058} C_VEL
LIN {X 0,Y 16.992,Z 828.07,A -85,B 0,C 180,E1 -31282.472,E2 -31282.472} C_VEL
LIN {X 0,Y 19.359,Z 838.54,A -85,B 0,C 180,E1 -31319.998,E2 -31319.998} C_VEL
LIN {X 0,Y 27.404,Z 847.323,A -85,B 0,C 180,E1 -31342.623,E2 -31342.623} C_VEL
LIN {X 0,Y 30.701,Z 849.875,A -85,B 0,C 180,E1 -31347.246,E2 -31347.246} C_VEL
LIN {X 0,Y 27.337,Z 848.544,A -85,B 0,C 180,E1 -31359.529,E2 -31359.529} C_VEL
LIN {X 0,Y 23.262,Z 844.255,A -85,B 0,C 180,E1 -31385.003,E2 -31385.003} C_VEL
LIN {X 0,Y 22.56,Z 842.724,A -85,B 0,C 180,E1 -31391.847,E2 -31391.847} C_VEL
LIN {X 0,Y 20.069,Z 835.848,A -85,B 0,C 180,E1 -31415.02,E2 -31415.02} C_VEL
LIN {X 0,Y 18.927,Z 826.833,A -85,B 0,C 180,E1 -31440.698,E2 -31440.698} C_VEL
LIN {X 0,Y 21.106,Z 815.236,A -85,B 0,C 180,E1 -31466.351,E2 -31466.351} C_VEL
LIN {X 0,Y 25.044,Z 803.557,A -85,B 0,C 180,E1 -31481.929,E2 -31481.929} C_VEL
LIN {X 0,Y 25.443,Z 802.456,A -85,B 0,C 180,E1 -31483.012,E2 -31483.012} C_VEL
LIN {X 0,Y 25.765,Z 800.279,A -85,B 0,C 180,E1 -31485.961,E2 -31485.961} C_VEL
LIN {X 0,Y 25.231,Z 797.962,A -85,B 0,C 180,E1 -31491.085,E2 -31491.085} C_VEL
LIN {X 0,Y 24.184,Z 796.159,A -85,B 0,C 180,E1 -31497.376,E2 -31497.376} C_VEL
LIN {X 0,Y 22.632,Z 794.612,A -85,B 0,C 180,E1 -31506.837,E2 -31506.837} C_VEL
LIN {X 0,Y 21.04,Z 793.424,A -85,B 0,C 180,E1 -31522.143,E2 -31522.143} C_VEL
LIN {X 0,Y 20.665,Z 793.206,A -85,B 0,C 180,E1 -31530.522,E2 -31530.522} C_VEL
LIN {X 0,Y 20.823,Z 793.073,A -85,B 0,C 180,E1 -31542.459,E2 -31542.459} C_VEL
LIN {X 0,Y 21.411,Z 796.323,A -85,B 0,C 180,E1 -31564.044,E2 -31564.044} C_VEL
LIN {X 0,Y 21.535,Z 797.26,A -85,B 0,C 180,E1 -31567.62,E2 -31567.62} C_VEL
LIN {X 0,Y 20.779,Z 804.223,A -85,B 0,C 180,E1 -31583.262,E2 -31583.262} C_VEL
LIN {X 0,Y 20.433,Z 806.407,A -85,B 0,C 180,E1 -31587.722,E2 -31587.722} C_VEL
LIN {X 0,Y 12.877,Z 819.022,A -85,B 0,C 180,E1 -31609.694,E2 -31609.694} C_VEL
LIN {X 0,Y 10.084,Z 829.617,A -85,B 0,C 180,E1 -31659.601,E2 -31659.601} C_VEL
LIN {X 0,Y 15.486,Z 838.607,A -85,B 0,C 180,E1 -31700.617,E2 -31700.617} C_VEL
LIN {X 0,Y 21.712,Z 844.288,A -85,B 0,C 180,E1 -31713.474,E2 -31713.474} C_VEL
LIN {X 0,Y 17.749,Z 840.897,A -85,B 0,C 180,E1 -31736.37,E2 -31736.37} C_VEL
LIN {X 0,Y 16.3,Z 839.083,A -85,B 0,C 180,E1 -31744.456,E2 -31744.456} C_VEL
LIN {X 0,Y 13.904,Z 834.673,A -85,B 0,C 180,E1 -31763.46,E2 -31763.46} C_VEL
LIN {X 0,Y 11.876,Z 825.861,A -85,B 0,C 180,E1 -31801.182,E2 -31801.182} C_VEL
LIN {X 0,Y 15.114,Z 814.281,A -85,B 0,C 180,E1 -31838.428,E2 -31838.428} C_VEL
LIN {X 0,Y 20.476,Z 802.352,A -85,B 0,C 180,E1 -31855.742,E2 -31855.742} C_VEL
LIN {X 0,Y 21.513,Z 800.041,A -85,B 0,C 180,E1 -31857.896,E2 -31857.896} C_VEL
LIN {X 0,Y 21.753,Z 796.787,A -85,B 0,C 180,E1 -31864.964,E2 -31864.964} C_VEL
LIN {X 0,Y 21.624,Z 794.423,A -85,B 0,C 180,E1 -31872.837,E2 -31872.837} C_VEL
LIN {X 0,Y 21.364,Z 793.336,A -85,B 0,C 180,E1 -31879.209,E2 -31879.209} C_VEL
LIN {X 0,Y 20.665,Z 793.206,A -85,B 0,C 180,E1 -31890.522,E2 -31890.522} C_VEL
LIN {X 0,Y 20.363,Z 793.712,A -85,B 0,C 180,E1 -31897.917,E2 -31897.917} C_VEL
LIN {X 0,Y 19.793,Z 795.47,A -85,B 0,C 180,E1 -31906.298,E2 -31906.298} C_VEL
LIN {X 0,Y 19.011,Z 797.947,A -85,B 0,C 180,E1 -31913.626,E2 -31913.626} C_VEL
LIN {X 0,Y 17.696,Z 801.59,A -85,B 0,C 180,E1 -31921.232,E2 -31921.232} C_VEL
LIN {X 0,Y 15.927,Z 805.539,A -85,B 0,C 180,E1 -31927.687,E2 -31927.687} C_VEL
LIN {X 0,Y 13.632,Z 809.404,A -85,B 0,C 180,E1 -31932.052,E2 -31932.052} C_VEL
LIN {X 0,Y 6.108,Z 819.629,A -85,B 0,C 180,E1 -31950.007,E2 -31950.007} C_VEL
LIN {X 0,Y 4.887,Z 829.249,A -85,B 0,C 180,E1 -32061.085,E2 -32061.085} C_VEL
LIN {X 0,Y 10.237,Z 834.786,A -85,B 0,C 180,E1 -32083.352,E2 -32083.352} C_VEL
LIN {X 0,Y 10.682,Z 835.105,A -85,B 0,C 180,E1 -32088.85,E2 -32088.85} C_VEL
LIN {X 0,Y 7.764,Z 831.686,A -85,B 0,C 180,E1 -32104.839,E2 -32104.839} C_VEL
LIN {X 0,Y 5.35,Z 822.353,A -85,B 0,C 180,E1 -32185.172,E2 -32185.172} C_VEL
LIN {X 0,Y 11.622,Z 811.306,A -85,B 0,C 180,E1 -32225.727,E2 -32225.727} C_VEL
LIN {X 0,Y 16.908,Z 802.183,A -85,B 0,C 180,E1 -32234.639,E2 -32234.639} C_VEL
LIN {X 0,Y 17.441,Z 801.044,A -85,B 0,C 180,E1 -32235.99,E2 -32235.99} C_VEL
LIN {X 0,Y 17.662,Z 799.542,A -85,B 0,C 180,E1 -32243.45,E2 -32243.45} C_VEL
LIN {X 0,Y 17.313,Z 799.434,A -85,B 0,C 180,E1 -32255.723,E2 -32255.723} C_VEL
LIN {X 0,Y 17.192,Z 801.239,A -85,B 0,C 180,E1 -32274.849,E2 -32274.849} C_VEL
LIN {X 0,Y 15.782,Z 805.779,A -85,B 0,C 180,E1 -32287.839,E2 -32287.839} C_VEL
LIN {X 0,Y 14.879,Z 807.599,A -85,B 0,C 180,E1 -32290.859,E2 -32290.859} C_VEL
LIN {X 0,Y 13.632,Z 809.404,A -85,B 0,C 180,E1 -32292.052,E2 -32292.052} C_VEL
LIN {X 0,Y 13.632,Z 809.404,A -85,B 0,C 180,E1 -32292.052,E2 -32292.052}

QRS_NEXT_CUT()

QRS_NEXT()
QRS_HOME()

END
